LIN {X -0.008,Y -156.128,Z 1901.908,A 0.000,B 0.000,C 90.000,E1 343.378} C_DIS
LIN {X 0.025,Y -158.540,Z 1901.883,A 0.000,B 0.000,C 90.000,E1 338.901} C_DIS
LIN {X 0.039,Y -162.151,Z 1901.858,A 0.000,B 0.000,C 90.000,E1 334.460} C_DIS
LIN {X 0.090,Y -166.092,Z 1901.839,A 0.000,B 0.000,C 90.000,E1 330.923} C_DIS
LIN {X 0.023,Y -169.681,Z 1901.824,A 0.000,B 0.000,C 90.000,E1 328.329} C_DIS
LIN {X 0.058,Y -173.811,Z 1901.810,A 0.000,B 0.000,C 90.000,E1 325.722} C_DIS
LIN {X -0.019,Y -178.557,Z 1901.795,A 0.000,B 0.000,C 90.000,E1 323.176} C_DIS
LIN {X -0.047,Y -184.121,Z 1901.781,A 0.000,B 0.000,C 90.000,E1 320.642} C_DIS
LIN {X 0.007,Y -190.588,Z 1901.767,A 0.000,B 0.000,C 90.000,E1 318.119} C_DIS
LIN {X 0.021,Y -198.074,Z 1901.754,A 0.000,B 0.000,C 90.000,E1 315.648} C_DIS
LIN {X 0.040,Y -206.500,Z 1901.740,A 0.000,B 0.000,C 90.000,E1 313.218} C_DIS
LIN {X -0.005,Y -217.446,Z 1901.725,A 0.000,B 0.000,C 90.000,E1 310.458} C_DIS
LIN {X 0.024,Y -231.204,Z 1901.708,A 0.000,B 0.000,C 90.000,E1 307.363} C_DIS
LIN {X -0.156,Y -246.156,Z 1901.691,A 0.000,B 0.000,C 90.000,E1 304.405} C_DIS
LIN {X -0.150,Y -258.005,Z 1901.679,A 0.000,B 0.000,C 90.000,E1 302.212} C_DIS
LIN {X 0.093,Y -272.069,Z 1901.665,A 0.000,B 0.000,C 90.000,E1 299.667} C_DIS
LIN {X -0.131,Y -281.961,Z 1901.655,A 0.000,B 0.000,C 90.000,E1 297.975} C_DIS
LIN {X 0.044,Y -291.566,Z 1901.646,A 0.000,B 0.000,C 90.000,E1 296.232} C_DIS
LIN {X -0.014,Y -298.859,Z 1901.638,A 0.000,B 0.000,C 90.000,E1 294.899} C_DIS
LIN {X 0.154,Y -306.333,Z 1901.633,A 0.000,B 0.000,C 90.000,E1 293.823} C_DIS
LIN {X 0.160,Y -315.202,Z 1901.625,A 0.000,B 0.000,C 90.000,E1 292.514} C_DIS
LIN {X -0.072,Y -321.527,Z 1901.620,A 0.000,B 0.000,C 90.000,E1 291.589} C_DIS
LIN {X 0.003,Y -329.446,Z 1901.613,A 0.000,B 0.000,C 90.000,E1 290.301} C_DIS
LIN {X 0.047,Y -338.650,Z 1901.604,A 0.000,B 0.000,C 90.000,E1 288.725} C_DIS
LIN {X -0.090,Y -343.776,Z 1901.599,A 0.000,B 0.000,C 90.000,E1 287.819} C_DIS
LIN {X 0.146,Y -348.475,Z 1901.594,A 0.000,B 0.000,C 90.000,E1 286.858} C_DIS
LIN {X -0.001,Y -352.501,Z 1901.589,A 0.000,B 0.000,C 90.000,E1 285.969} C_DIS
LIN {X -0.022,Y -355.999,Z 1901.584,A 0.000,B 0.000,C 90.000,E1 285.064} C_DIS
LIN {X -0.140,Y -358.008,Z 1901.580,A 0.000,B 0.000,C 90.000,E1 284.481} C_DIS
LIN {X -0.161,Y -359.770,Z 1901.577,A 0.000,B 0.000,C 90.000,E1 283.883} C_DIS
LIN {X 0.094,Y -361.166,Z 1901.574,A 0.000,B 0.000,C 90.000,E1 283.244} C_DIS
LIN {X 0.093,Y -362.224,Z 1901.570,A 0.000,B 0.000,C 90.000,E1 282.647} C_DIS
LIN {X 0.017,Y -362.868,Z 1901.567,A 0.000,B 0.000,C 90.000,E1 282.063} C_DIS
LIN {X -0.050,Y -363.124,Z 1901.564,A 0.000,B 0.000,C 90.000,E1 281.478} C_DIS
LIN {X -0.113,Y -363.007,Z 1901.560,A 0.000,B 0.000,C 90.000,E1 280.894} C_DIS
LIN {X 0.182,Y -362.489,Z 1901.557,A 0.000,B 0.000,C 90.000,E1 280.254} C_DIS
LIN {X 0.117,Y -361.578,Z 1901.554,A 0.000,B 0.000,C 90.000,E1 279.670} C_DIS
LIN {X -0.008,Y -360.355,Z 1901.551,A 0.000,B 0.000,C 90.000,E1 279.095} C_DIS
LIN {X -0.081,Y -358.715,Z 1901.547,A 0.000,B 0.000,C 90.000,E1 278.511} C_DIS
LIN {X 0.093,Y -355.791,Z 1901.542,A 0.000,B 0.000,C 90.000,E1 277.587} C_DIS
LIN {X -0.112,Y -351.986,Z 1901.537,A 0.000,B 0.000,C 90.000,E1 276.720} C_DIS
LIN {X -0.007,Y -347.191,Z 1901.532,A 0.000,B 0.000,C 90.000,E1 275.796} C_DIS
LIN {X 0.141,Y -343.273,Z 1901.529,A 0.000,B 0.000,C 90.000,E1 275.163} C_DIS
LIN {X -0.075,Y -338.789,Z 1901.525,A 0.000,B 0.000,C 90.000,E1 274.588} C_DIS
LIN {X 0.022,Y -333.591,Z 1901.522,A 0.000,B 0.000,C 90.000,E1 273.955} C_DIS
LIN {X -0.141,Y -327.774,Z 1901.519,A 0.000,B 0.000,C 90.000,E1 273.383} C_DIS
LIN {X -0.062,Y -321.579,Z 1901.516,A 0.000,B 0.000,C 90.000,E1 272.808} C_DIS
LIN {X -0.009,Y -315.100,Z 1901.513,A 0.000,B 0.000,C 90.000,E1 272.293} C_DIS
LIN {X 0.118,Y -308.269,Z 1901.510,A 0.000,B 0.000,C 90.000,E1 271.835} C_DIS
LIN {X 0.007,Y -301.029,Z 1901.508,A 0.000,B 0.000,C 90.000,E1 271.489} C_DIS
LIN {X -0.028,Y -293.012,Z 1901.507,A 0.000,B 0.000,C 90.000,E1 271.203} C_DIS
LIN {X -0.091,Y -287.800,Z 1901.506,A 0.000,B 0.000,C 90.000,E1 271.088} C_DIS
LIN {X -0.114,Y -278.697,Z 1901.505,A 0.000,B 0.000,C 90.000,E1 270.974} C_DIS
LIN {X -0.029,Y -270.235,Z 1901.505,A 0.000,B 0.000,C 90.000,E1 270.917} C_DIS
LIN {X -0.041,Y -181.478,Z 1901.505,A 0.000,B 0.000,C 90.000,E1 270.917} C_DIS
LIN {X -0.028,Y -181.537,Z 1901.499,A 0.000,B 0.000,C 90.000,E1 269.885} C_DIS
LIN {X -0.085,Y -180.907,Z 1901.475,A 0.000,B 0.000,C 90.000,E1 265.527} C_DIS
LIN {X -0.027,Y -180.749,Z 1901.470,A 0.000,B 0.000,C 90.000,E1 264.666} C_DIS
LIN {X 0.041,Y -178.842,Z 1901.442,A 0.000,B 0.000,C 90.000,E1 259.577} C_DIS
LIN {X -0.063,Y -175.885,Z 1901.414,A 0.000,B 0.000,C 90.000,E1 254.519} C_DIS
LIN {X 0.044,Y -174.552,Z 1901.404,A 0.000,B 0.000,C 90.000,E1 252.779} C_DIS
LIN {X -0.025,Y -171.536,Z 1901.381,A 0.000,B 0.000,C 90.000,E1 248.518} C_DIS
LIN {X -0.031,Y -167.761,Z 1901.357,A 0.000,B 0.000,C 90.000,E1 244.204} C_DIS
LIN {X -0.088,Y -166.467,Z 1901.347,A 0.000,B 0.000,C 90.000,E1 242.487} C_DIS
LIN {X 0.048,Y -163.182,Z 1901.328,A 0.000,B 0.000,C 90.000,E1 238.948} C_DIS
LIN {X -0.037,Y -161.142,Z 1901.313,A 0.000,B 0.000,C 90.000,E1 236.342} C_DIS
LIN {X -0.001,Y -157.162,Z 1901.288,A 0.000,B 0.000,C 90.000,E1 231.904} C_DIS
LIN {X 0.022,Y -155.893,Z 1901.278,A 0.000,B 0.000,C 90.000,E1 230.114} C_DIS
LIN {X -0.020,Y -152.144,Z 1901.254,A 0.000,B 0.000,C 90.000,E1 225.648} C_DIS
LIN {X 0.000,Y -150.393,Z 1901.239,A 0.000,B 0.000,C 90.000,E1 222.933} C_DIS
LIN {X 0.024,Y -147.124,Z 1901.213,A 0.000,B 0.000,C 90.000,E1 218.382} C_DIS
LIN {X 0.015,Y -145.687,Z 1901.198,A 0.000,B 0.000,C 90.000,E1 215.644} C_DIS
LIN {X 0.013,Y -143.070,Z 1901.172,A 0.000,B 0.000,C 90.000,E1 211.052} C_DIS
LIN {X -0.056,Y -141.691,Z 1901.152,A 0.000,B 0.000,C 90.000,E1 207.385} C_DIS
LIN {X -0.002,Y -139.462,Z 1901.116,A 0.000,B 0.000,C 90.000,E1 200.865} C_DIS
LIN {X -0.033,Y -139.195,Z 1901.106,A 0.000,B 0.000,C 90.000,E1 199.014} C_DIS
LIN {X -0.015,Y -138.326,Z 1901.054,A 0.000,B 0.000,C 90.000,E1 189.670} C_DIS
LIN {X -0.010,Y -139.451,Z 1901.007,A 0.000,B 0.000,C 90.000,E1 181.260} C_DIS
LIN {X 0.070,Y -140.996,Z 1900.976,A 0.000,B 0.000,C 90.000,E1 175.641} C_DIS
LIN {X 0.020,Y -142.749,Z 1900.955,A 0.000,B 0.000,C 90.000,E1 171.951} C_DIS
LIN {X -0.024,Y -145.149,Z 1900.930,A 0.000,B 0.000,C 90.000,E1 167.353} C_DIS
LIN {X -0.031,Y -147.771,Z 1900.909,A 0.000,B 0.000,C 90.000,E1 163.685} C_DIS
LIN {X 0.049,Y -150.447,Z 1900.889,A 0.000,B 0.000,C 90.000,E1 160.007} C_DIS
LIN {X -0.017,Y -153.894,Z 1900.869,A 0.000,B 0.000,C 90.000,E1 156.410} C_DIS
LIN {X -0.023,Y -157.305,Z 1900.849,A 0.000,B 0.000,C 90.000,E1 152.820} C_DIS
LIN {X -0.004,Y -161.490,Z 1900.829,A 0.000,B 0.000,C 90.000,E1 149.253} C_DIS
LIN {X 0.011,Y -165.689,Z 1900.810,A 0.000,B 0.000,C 90.000,E1 145.722} C_DIS
LIN {X -0.102,Y -170.631,Z 1900.790,A 0.000,B 0.000,C 90.000,E1 142.271} C_DIS
LIN {X 0.052,Y -175.508,Z 1900.771,A 0.000,B 0.000,C 90.000,E1 138.771} C_DIS
LIN {X -0.082,Y -181.129,Z 1900.752,A 0.000,B 0.000,C 90.000,E1 135.405} C_DIS
LIN {X 0.045,Y -186.577,Z 1900.733,A 0.000,B 0.000,C 90.000,E1 132.000} C_DIS
LIN {X -0.006,Y -191.189,Z 1900.719,A 0.000,B 0.000,C 90.000,E1 129.519} C_DIS
LIN {X 0.040,Y -196.998,Z 1900.701,A 0.000,B 0.000,C 90.000,E1 126.217} C_DIS
LIN {X -0.042,Y -200.267,Z 1900.692,A 0.000,B 0.000,C 90.000,E1 124.612} C_DIS
LIN {X -0.049,Y -207.759,Z 1900.670,A 0.000,B 0.000,C 90.000,E1 120.590} C_DIS
LIN {X -0.046,Y -210.934,Z 1900.661,A 0.000,B 0.000,C 90.000,E1 118.999} C_DIS
LIN {X -0.040,Y -216.804,Z 1900.644,A 0.000,B 0.000,C 90.000,E1 115.848} C_DIS
LIN {X 0.108,Y -218.419,Z 1900.639,A 0.000,B 0.000,C 90.000,E1 115.027} C_DIS
LIN {X -0.053,Y -221.146,Z 1900.631,A 0.000,B 0.000,C 90.000,E1 113.515} C_DIS
LIN {X -0.062,Y -224.140,Z 1900.621,A 0.000,B 0.000,C 90.000,E1 111.844} C_DIS
LIN {X -0.111,Y -283.670,Z 1900.621,A 0.000,B 0.000,C 90.000,E1 111.844} C_DIS
LIN {X 0.092,Y -285.624,Z 1900.621,A 0.000,B 0.000,C 90.000,E1 111.770} C_DIS
LIN {X 0.027,Y -291.063,Z 1900.619,A 0.000,B 0.000,C 90.000,E1 111.482} C_DIS
LIN {X 0.066,Y -293.925,Z 1900.618,A 0.000,B 0.000,C 90.000,E1 111.173} C_DIS
LIN {X -0.146,Y -295.977,Z 1900.616,A 0.000,B 0.000,C 90.000,E1 110.918} C_DIS
LIN {X -0.054,Y -310.986,Z 1900.602,A 0.000,B 0.000,C 90.000,E1 108.290} C_DIS
LIN {X -0.018,Y -325.732,Z 1900.589,A 0.000,B 0.000,C 90.000,E1 106.024} C_DIS
LIN {X 0.068,Y -339.562,Z 1900.578,A 0.000,B 0.000,C 90.000,E1 104.120} C_DIS
LIN {X -0.082,Y -354.591,Z 1900.568,A 0.000,B 0.000,C 90.000,E1 102.299} C_DIS
LIN {X 0.090,Y -373.026,Z 1900.557,A 0.000,B 0.000,C 90.000,E1 100.254} C_DIS
LIN {X -0.167,Y -391.934,Z 1900.547,A 0.000,B 0.000,C 90.000,E1 98.454} C_DIS
LIN {X -0.127,Y -411.181,Z 1900.538,A 0.000,B 0.000,C 90.000,E1 96.777} C_DIS
LIN {X -0.181,Y -433.588,Z 1900.528,A 0.000,B 0.000,C 90.000,E1 95.049} C_DIS
LIN {X -0.202,Y -439.236,Z 1900.526,A 0.000,B 0.000,C 90.000,E1 94.645} C_DIS
LIN {X 0.011,Y -441.525,Z 1900.525,A 0.000,B 0.000,C 90.000,E1 94.416} C_DIS
LIN {X -0.022,Y -445.053,Z 1900.522,A 0.000,B 0.000,C 90.000,E1 93.955} C_DIS
LIN {X 0.151,Y -446.391,Z 1900.521,A 0.000,B 0.000,C 90.000,E1 93.669} C_DIS
LIN {X -0.120,Y -447.386,Z 1900.519,A 0.000,B 0.000,C 90.000,E1 93.440} C_DIS
LIN {X -0.163,Y -448.538,Z 1900.516,A 0.000,B 0.000,C 90.000,E1 92.922} C_DIS
LIN {X -0.223,Y -448.727,Z 1900.513,A 0.000,B 0.000,C 90.000,E1 92.407} C_DIS
LIN {X 0.176,Y -447.984,Z 1900.510,A 0.000,B 0.000,C 90.000,E1 91.835} C_DIS
LIN {X 0.140,Y -446.197,Z 1900.507,A 0.000,B 0.000,C 90.000,E1 91.318} C_DIS
LIN {X -0.109,Y -444.813,Z 1900.506,A 0.000,B 0.000,C 90.000,E1 91.088} C_DIS
LIN {X -0.021,Y -431.659,Z 1900.494,A 0.000,B 0.000,C 90.000,E1 88.969} C_DIS
LIN {X -0.041,Y -421.590,Z 1900.485,A 0.000,B 0.000,C 90.000,E1 87.364} C_DIS
LIN {X -0.125,Y -409.813,Z 1900.475,A 0.000,B 0.000,C 90.000,E1 85.469} C_DIS
LIN {X -0.057,Y -399.632,Z 1900.465,A 0.000,B 0.000,C 90.000,E1 83.799} C_DIS
LIN {X -0.119,Y -387.656,Z 1900.455,A 0.000,B 0.000,C 90.000,E1 81.837} C_DIS
LIN {X 0.076,Y -374.093,Z 1900.442,A 0.000,B 0.000,C 90.000,E1 79.511} C_DIS
LIN {X -0.009,Y -356.071,Z 1900.424,A 0.000,B 0.000,C 90.000,E1 76.284} C_DIS
LIN {X 0.010,Y -342.262,Z 1900.409,A 0.000,B 0.000,C 90.000,E1 73.559} C_DIS
LIN {X -0.031,Y -330.388,Z 1900.395,A 0.000,B 0.000,C 90.000,E1 71.094} C_DIS
LIN {X 0.098,Y -317.360,Z 1900.379,A 0.000,B 0.000,C 90.000,E1 68.230} C_DIS
LIN {X -0.076,Y -304.962,Z 1900.363,A 0.000,B 0.000,C 90.000,E1 65.357} C_DIS
LIN {X -0.057,Y -295.446,Z 1900.350,A 0.000,B 0.000,C 90.000,E1 63.050} C_DIS
LIN {X -0.111,Y -286.135,Z 1900.337,A 0.000,B 0.000,C 90.000,E1 60.717} C_DIS
LIN {X -0.085,Y -276.695,Z 1900.324,A 0.000,B 0.000,C 90.000,E1 58.329} C_DIS
LIN {X 0.012,Y -267.201,Z 1900.310,A 0.000,B 0.000,C 90.000,E1 55.881} C_DIS
LIN {X -0.020,Y -257.579,Z 1900.297,A 0.000,B 0.000,C 90.000,E1 53.417} C_DIS
LIN {X 0.042,Y -247.984,Z 1900.283,A 0.000,B 0.000,C 90.000,E1 50.884} C_DIS
LIN {X -0.005,Y -237.137,Z 1900.266,A 0.000,B 0.000,C 90.000,E1 47.957} C_DIS
LIN {X -0.021,Y -226.676,Z 1900.250,A 0.000,B 0.000,C 90.000,E1 44.960} C_DIS
LIN {X -0.056,Y -215.454,Z 1900.231,A 0.000,B 0.000,C 90.000,E1 41.515} C_DIS
LIN {X -0.080,Y -206.223,Z 1900.213,A 0.000,B 0.000,C 90.000,E1 38.382} C_DIS
LIN {X -0.068,Y -197.894,Z 1900.195,A 0.000,B 0.000,C 90.000,E1 35.185} C_DIS
LIN {X -0.046,Y -190.289,Z 1900.177,A 0.000,B 0.000,C 90.000,E1 31.926} C_DIS
LIN {X -0.030,Y -183.438,Z 1900.159,A 0.000,B 0.000,C 90.000,E1 28.615} C_DIS
LIN {X -0.113,Y -177.266,Z 1900.140,A 0.000,B 0.000,C 90.000,E1 25.283} C_DIS
LIN {X -0.007,Y -171.928,Z 1900.121,A 0.000,B 0.000,C 90.000,E1 21.844} C_DIS
LIN {X -0.067,Y -167.365,Z 1900.102,A 0.000,B 0.000,C 90.000,E1 18.417} C_DIS
LIN {X 0.033,Y -163.638,Z 1900.083,A 0.000,B 0.000,C 90.000,E1 14.898} C_DIS
LIN {X 0.064,Y -159.841,Z 1900.058,A 0.000,B 0.000,C 90.000,E1 10.489} C_DIS
LIN {X -0.028,Y -157.203,Z 1900.034,A 0.000,B 0.000,C 90.000,E1 6.087} C_DIS
LIN {X 0.000,Y -154.884,Z 1900.000,A 0.000,B 0.000,C 90.000,E1 360.000} C_DIS
LIN {X -0.012,Y -154.116,Z 1899.948,A 0.000,B 0.000,C 90.000,E1 350.557} C_DIS
LIN {X -0.008,Y -156.124,Z 1899.908,A 0.000,B 0.000,C 90.000,E1 343.378} C_DIS
LIN {X 0.025,Y -158.536,Z 1899.883,A 0.000,B 0.000,C 90.000,E1 338.901} C_DIS
LIN {X 0.038,Y -162.149,Z 1899.858,A 0.000,B 0.000,C 90.000,E1 334.460} C_DIS
LIN {X 0.089,Y -166.095,Z 1899.839,A 0.000,B 0.000,C 90.000,E1 330.923} C_DIS
LIN {X 0.023,Y -169.685,Z 1899.824,A 0.000,B 0.000,C 90.000,E1 328.329} C_DIS
LIN {X 0.056,Y -173.818,Z 1899.810,A 0.000,B 0.000,C 90.000,E1 325.722} C_DIS
LIN {X -0.019,Y -178.565,Z 1899.795,A 0.000,B 0.000,C 90.000,E1 323.176} C_DIS
LIN {X -0.047,Y -184.128,Z 1899.781,A 0.000,B 0.000,C 90.000,E1 320.642} C_DIS
LIN {X 0.007,Y -190.596,Z 1899.767,A 0.000,B 0.000,C 90.000,E1 318.119} C_DIS
LIN {X 0.020,Y -198.081,Z 1899.754,A 0.000,B 0.000,C 90.000,E1 315.648} C_DIS
LIN {X 0.040,Y -206.507,Z 1899.740,A 0.000,B 0.000,C 90.000,E1 313.218} C_DIS
LIN {X -0.005,Y -217.454,Z 1899.725,A 0.000,B 0.000,C 90.000,E1 310.458} C_DIS
LIN {X 0.024,Y -231.213,Z 1899.708,A 0.000,B 0.000,C 90.000,E1 307.363} C_DIS
LIN {X -0.155,Y -246.166,Z 1899.691,A 0.000,B 0.000,C 90.000,E1 304.405} C_DIS
LIN {X -0.150,Y -258.015,Z 1899.679,A 0.000,B 0.000,C 90.000,E1 302.212} C_DIS
LIN {X 0.093,Y -272.077,Z 1899.665,A 0.000,B 0.000,C 90.000,E1 299.667} C_DIS
LIN {X -0.130,Y -281.970,Z 1899.655,A 0.000,B 0.000,C 90.000,E1 297.975} C_DIS
LIN {X 0.045,Y -291.575,Z 1899.646,A 0.000,B 0.000,C 90.000,E1 296.232} C_DIS
LIN {X -0.129,Y -295.469,Z 1899.642,A 0.000,B 0.000,C 90.000,E1 295.591} C_DIS
LIN {X 0.060,Y -305.331,Z 1899.634,A 0.000,B 0.000,C 90.000,E1 294.131} C_DIS
LIN {X 0.048,Y -313.975,Z 1899.627,A 0.000,B 0.000,C 90.000,E1 292.823} C_DIS
LIN {X 0.029,Y -322.355,Z 1899.620,A 0.000,B 0.000,C 90.000,E1 291.535} C_DIS
LIN {X 0.119,Y -330.255,Z 1899.613,A 0.000,B 0.000,C 90.000,E1 290.248} C_DIS
LIN {X -0.139,Y -339.493,Z 1899.604,A 0.000,B 0.000,C 90.000,E1 288.725} C_DIS
LIN {X 0.057,Y -344.603,Z 1899.599,A 0.000,B 0.000,C 90.000,E1 287.764} C_DIS
LIN {X -0.037,Y -347.799,Z 1899.595,A 0.000,B 0.000,C 90.000,E1 287.166} C_DIS
LIN {X -0.097,Y -351.986,Z 1899.590,A 0.000,B 0.000,C 90.000,E1 286.260} C_DIS
LIN {X 0.129,Y -355.611,Z 1899.585,A 0.000,B 0.000,C 90.000,E1 285.315} C_DIS
LIN {X 0.047,Y -358.698,Z 1899.580,A 0.000,B 0.000,C 90.000,E1 284.426} C_DIS
LIN {X 0.031,Y -360.418,Z 1899.577,A 0.000,B 0.000,C 90.000,E1 283.828} C_DIS
LIN {X -0.059,Y -361.770,Z 1899.573,A 0.000,B 0.000,C 90.000,E1 283.244} C_DIS
LIN {X -0.057,Y -362.810,Z 1899.570,A 0.000,B 0.000,C 90.000,E1 282.647} C_DIS
LIN {X -0.129,Y -363.440,Z 1899.567,A 0.000,B 0.000,C 90.000,E1 282.063} C_DIS
LIN {X 0.164,Y -363.653,Z 1899.564,A 0.000,B 0.000,C 90.000,E1 281.422} C_DIS
LIN {X 0.104,Y -363.520,Z 1899.560,A 0.000,B 0.000,C 90.000,E1 280.838} C_DIS
LIN {X 0.045,Y -362.940,Z 1899.557,A 0.000,B 0.000,C 90.000,E1 280.254} C_DIS
LIN {X -0.015,Y -361.997,Z 1899.554,A 0.000,B 0.000,C 90.000,E1 279.670} C_DIS
LIN {X -0.138,Y -360.713,Z 1899.550,A 0.000,B 0.000,C 90.000,E1 279.095} C_DIS
LIN {X 0.147,Y -359.050,Z 1899.547,A 0.000,B 0.000,C 90.000,E1 278.454} C_DIS
LIN {X -0.029,Y -356.047,Z 1899.542,A 0.000,B 0.000,C 90.000,E1 277.587} C_DIS
LIN {X 0.120,Y -352.226,Z 1899.537,A 0.000,B 0.000,C 90.000,E1 276.663} C_DIS
LIN {X -0.122,Y -347.361,Z 1899.532,A 0.000,B 0.000,C 90.000,E1 275.796} C_DIS
LIN {X 0.029,Y -343.402,Z 1899.529,A 0.000,B 0.000,C 90.000,E1 275.163} C_DIS
LIN {X 0.153,Y -338.870,Z 1899.525,A 0.000,B 0.000,C 90.000,E1 274.531} C_DIS
LIN {X -0.084,Y -333.652,Z 1899.522,A 0.000,B 0.000,C 90.000,E1 273.955} C_DIS
LIN {X 0.106,Y -327.877,Z 1899.519,A 0.000,B 0.000,C 90.000,E1 273.326} C_DIS
LIN {X -0.085,Y -321.739,Z 1899.516,A 0.000,B 0.000,C 90.000,E1 272.808} C_DIS
LIN {X -0.012,Y -315.422,Z 1899.513,A 0.000,B 0.000,C 90.000,E1 272.293} C_DIS
LIN {X 0.059,Y -308.778,Z 1899.510,A 0.000,B 0.000,C 90.000,E1 271.835} C_DIS
LIN {X 0.150,Y -301.714,Z 1899.508,A 0.000,B 0.000,C 90.000,E1 271.432} C_DIS
LIN {X -0.007,Y -294.014,Z 1899.506,A 0.000,B 0.000,C 90.000,E1 271.146} C_DIS
LIN {X -0.027,Y -284.992,Z 1899.505,A 0.000,B 0.000,C 90.000,E1 270.917} C_DIS
LIN {X 0.132,Y -275.226,Z 1899.504,A 0.000,B 0.000,C 90.000,E1 270.745} C_DIS
LIN {X 0.093,Y -264.382,Z 1899.504,A 0.000,B 0.000,C 90.000,E1 270.688} C_DIS
LIN {X 0.034,Y -181.526,Z 1899.504,A 0.000,B 0.000,C 90.000,E1 270.688} C_DIS
LIN {X 0.084,Y -181.487,Z 1899.498,A 0.000,B 0.000,C 90.000,E1 269.656} C_DIS
LIN {X 0.026,Y -180.904,Z 1899.474,A 0.000,B 0.000,C 90.000,E1 265.298} C_DIS
LIN {X -0.024,Y -180.247,Z 1899.465,A 0.000,B 0.000,C 90.000,E1 263.628} C_DIS
LIN {X -0.005,Y -178.736,Z 1899.441,A 0.000,B 0.000,C 90.000,E1 259.398} C_DIS
LIN {X 0.061,Y -175.784,Z 1899.413,A 0.000,B 0.000,C 90.000,E1 254.283} C_DIS
LIN {X 0.049,Y -171.968,Z 1899.384,A 0.000,B 0.000,C 90.000,E1 249.156} C_DIS
LIN {X 0.087,Y -171.366,Z 1899.380,A 0.000,B 0.000,C 90.000,E1 248.284} C_DIS
LIN {X -0.088,Y -167.614,Z 1899.355,A 0.000,B 0.000,C 90.000,E1 244.024} C_DIS
LIN {X 0.076,Y -166.263,Z 1899.346,A 0.000,B 0.000,C 90.000,E1 242.231} C_DIS
LIN {X 0.063,Y -163.016,Z 1899.326,A 0.000,B 0.000,C 90.000,E1 238.742} C_DIS
LIN {X -0.024,Y -160.940,Z 1899.312,A 0.000,B 0.000,C 90.000,E1 236.135} C_DIS
LIN {X 0.085,Y -157.698,Z 1899.292,A 0.000,B 0.000,C 90.000,E1 232.557} C_DIS
LIN {X 0.024,Y -155.738,Z 1899.277,A 0.000,B 0.000,C 90.000,E1 229.908} C_DIS
LIN {X 0.077,Y -151.996,Z 1899.252,A 0.000,B 0.000,C 90.000,E1 225.405} C_DIS
LIN {X 0.092,Y -150.241,Z 1899.237,A 0.000,B 0.000,C 90.000,E1 222.690} C_DIS
LIN {X 0.015,Y -147.000,Z 1899.212,A 0.000,B 0.000,C 90.000,E1 218.177} C_DIS
LIN {X 0.005,Y -145.584,Z 1899.197,A 0.000,B 0.000,C 90.000,E1 215.438} C_DIS
LIN {X -0.001,Y -142.973,Z 1899.171,A 0.000,B 0.000,C 90.000,E1 210.846} C_DIS
LIN {X 0.052,Y -141.600,Z 1899.151,A 0.000,B 0.000,C 90.000,E1 207.129} C_DIS
LIN {X -0.032,Y -139.423,Z 1899.115,A 0.000,B 0.000,C 90.000,E1 200.663} C_DIS
LIN {X 0.019,Y -139.150,Z 1899.104,A 0.000,B 0.000,C 90.000,E1 198.779} C_DIS
LIN {X 0.041,Y -138.344,Z 1899.058,A 0.000,B 0.000,C 90.000,E1 190.366} C_DIS
LIN {X 0.027,Y -139.486,Z 1899.006,A 0.000,B 0.000,C 90.000,E1 181.031} C_DIS
LIN {X -0.033,Y -141.084,Z 1898.975,A 0.000,B 0.000,C 90.000,E1 175.469} C_DIS
LIN {X 0.061,Y -142.461,Z 1898.959,A 0.000,B 0.000,C 90.000,E1 172.648} C_DIS
LIN {X 0.010,Y -144.706,Z 1898.934,A 0.000,B 0.000,C 90.000,E1 168.049} C_DIS
LIN {X -0.038,Y -147.303,Z 1898.913,A 0.000,B 0.000,C 90.000,E1 164.393} C_DIS
LIN {X -0.024,Y -150.624,Z 1898.888,A 0.000,B 0.000,C 90.000,E1 159.826} C_DIS
LIN {X 0.053,Y -154.099,Z 1898.868,A 0.000,B 0.000,C 90.000,E1 156.177} C_DIS
LIN {X -0.023,Y -157.522,Z 1898.848,A 0.000,B 0.000,C 90.000,E1 152.615} C_DIS
LIN {X -0.079,Y -161.756,Z 1898.828,A 0.000,B 0.000,C 90.000,E1 149.076} C_DIS
LIN {X 0.027,Y -165.949,Z 1898.808,A 0.000,B 0.000,C 90.000,E1 145.515} C_DIS
LIN {X 0.024,Y -170.940,Z 1898.789,A 0.000,B 0.000,C 90.000,E1 142.029} C_DIS
LIN {X -0.056,Y -175.809,Z 1898.770,A 0.000,B 0.000,C 90.000,E1 138.609} C_DIS
LIN {X 0.072,Y -181.416,Z 1898.751,A 0.000,B 0.000,C 90.000,E1 135.162} C_DIS
LIN {X -0.053,Y -186.918,Z 1898.732,A 0.000,B 0.000,C 90.000,E1 131.838} C_DIS
LIN {X 0.020,Y -191.497,Z 1898.719,A 0.000,B 0.000,C 90.000,E1 129.322} C_DIS
LIN {X 0.105,Y -197.361,Z 1898.700,A 0.000,B 0.000,C 90.000,E1 126.011} C_DIS
LIN {X 0.030,Y -200.637,Z 1898.691,A 0.000,B 0.000,C 90.000,E1 124.405} C_DIS
LIN {X -0.060,Y -206.521,Z 1898.673,A 0.000,B 0.000,C 90.000,E1 121.209} C_DIS
LIN {X 0.034,Y -209.811,Z 1898.664,A 0.000,B 0.000,C 90.000,E1 119.589} C_DIS
LIN {X -0.040,Y -217.169,Z 1898.643,A 0.000,B 0.000,C 90.000,E1 115.668} C_DIS
LIN {X -0.085,Y -218.796,Z 1898.638,A 0.000,B 0.000,C 90.000,E1 114.899} C_DIS
LIN {X -0.069,Y -224.144,Z 1898.621,A 0.000,B 0.000,C 90.000,E1 111.844} C_DIS
LIN {X -0.121,Y -284.036,Z 1898.621,A 0.000,B 0.000,C 90.000,E1 111.844} C_DIS
LIN {X 0.048,Y -285.983,Z 1898.621,A 0.000,B 0.000,C 90.000,E1 111.770} C_DIS
LIN {X 0.130,Y -289.404,Z 1898.620,A 0.000,B 0.000,C 90.000,E1 111.589} C_DIS
LIN {X 0.176,Y -292.839,Z 1898.618,A 0.000,B 0.000,C 90.000,E1 111.280} C_DIS
LIN {X 0.071,Y -296.478,Z 1898.616,A 0.000,B 0.000,C 90.000,E1 110.791} C_DIS
LIN {X -0.031,Y -309.743,Z 1898.603,A 0.000,B 0.000,C 90.000,E1 108.489} C_DIS
LIN {X 0.080,Y -324.361,Z 1898.590,A 0.000,B 0.000,C 90.000,E1 106.205} C_DIS
LIN {X 0.146,Y -338.072,Z 1898.580,A 0.000,B 0.000,C 90.000,E1 104.300} C_DIS
LIN {X -0.025,Y -352.972,Z 1898.569,A 0.000,B 0.000,C 90.000,E1 102.479} C_DIS
LIN {X 0.041,Y -371.365,Z 1898.558,A 0.000,B 0.000,C 90.000,E1 100.433} C_DIS
LIN {X 0.127,Y -390.236,Z 1898.548,A 0.000,B 0.000,C 90.000,E1 98.568} C_DIS
LIN {X 0.082,Y -409.450,Z 1898.538,A 0.000,B 0.000,C 90.000,E1 96.891} C_DIS
LIN {X -0.071,Y -431.829,Z 1898.529,A 0.000,B 0.000,C 90.000,E1 95.163} C_DIS
LIN {X 0.085,Y -440.191,Z 1898.525,A 0.000,B 0.000,C 90.000,E1 94.531} C_DIS
LIN {X -0.031,Y -443.932,Z 1898.523,A 0.000,B 0.000,C 90.000,E1 94.131} C_DIS
LIN {X 0.169,Y -445.542,Z 1898.521,A 0.000,B 0.000,C 90.000,E1 93.841} C_DIS
LIN {X -0.106,Y -446.756,Z 1898.520,A 0.000,B 0.000,C 90.000,E1 93.612} C_DIS
LIN {X -0.154,Y -448.257,Z 1898.517,A 0.000,B 0.000,C 90.000,E1 93.094} C_DIS
LIN {X -0.218,Y -448.753,Z 1898.514,A 0.000,B 0.000,C 90.000,E1 92.579} C_DIS
LIN {X 0.178,Y -448.320,Z 1898.511,A 0.000,B 0.000,C 90.000,E1 92.007} C_DIS
LIN {X 0.143,Y -446.901,Z 1898.508,A 0.000,B 0.000,C 90.000,E1 91.489} C_DIS
LIN {X -0.106,Y -445.751,Z 1898.507,A 0.000,B 0.000,C 90.000,E1 91.260} C_DIS
LIN {X 0.205,Y -439.284,Z 1898.501,A 0.000,B 0.000,C 90.000,E1 90.172} C_DIS
LIN {X -0.125,Y -429.425,Z 1898.492,A 0.000,B 0.000,C 90.000,E1 88.625} C_DIS
LIN {X -0.050,Y -417.625,Z 1898.482,A 0.000,B 0.000,C 90.000,E1 86.731} C_DIS
LIN {X 0.189,Y -405.837,Z 1898.471,A 0.000,B 0.000,C 90.000,E1 84.780} C_DIS
LIN {X -0.140,Y -393.895,Z 1898.460,A 0.000,B 0.000,C 90.000,E1 82.875} C_DIS
LIN {X 0.115,Y -381.954,Z 1898.449,A 0.000,B 0.000,C 90.000,E1 80.849} C_DIS
LIN {X 0.168,Y -368.450,Z 1898.436,A 0.000,B 0.000,C 90.000,E1 78.522} C_DIS
LIN {X 0.030,Y -352.386,Z 1898.420,A 0.000,B 0.000,C 90.000,E1 75.574} C_DIS
LIN {X 0.047,Y -338.733,Z 1898.405,A 0.000,B 0.000,C 90.000,E1 72.834} C_DIS
LIN {X -0.078,Y -326.939,Z 1898.391,A 0.000,B 0.000,C 90.000,E1 70.369} C_DIS
LIN {X -0.006,Y -312.664,Z 1898.373,A 0.000,B 0.000,C 90.000,E1 67.177} C_DIS
LIN {X -0.065,Y -301.772,Z 1898.359,A 0.000,B 0.000,C 90.000,E1 64.588} C_DIS
LIN {X -0.009,Y -289.633,Z 1898.342,A 0.000,B 0.000,C 90.000,E1 61.591} C_DIS
LIN {X 0.116,Y -281.614,Z 1898.331,A 0.000,B 0.000,C 90.000,E1 59.537} C_DIS
LIN {X -0.055,Y -272.131,Z 1898.318,A 0.000,B 0.000,C 90.000,E1 57.168} C_DIS
LIN {X 0.027,Y -263.959,Z 1898.306,A 0.000,B 0.000,C 90.000,E1 55.055} C_DIS
LIN {X 0.071,Y -254.351,Z 1898.292,A 0.000,B 0.000,C 90.000,E1 52.557} C_DIS
LIN {X 0.027,Y -244.761,Z 1898.278,A 0.000,B 0.000,C 90.000,E1 50.033} C_DIS
LIN {X 0.066,Y -233.998,Z 1898.262,A 0.000,B 0.000,C 90.000,E1 47.067} C_DIS
LIN {X 0.134,Y -223.664,Z 1898.245,A 0.000,B 0.000,C 90.000,E1 44.028} C_DIS
LIN {X -0.129,Y -212.650,Z 1898.225,A 0.000,B 0.000,C 90.000,E1 40.620} C_DIS
LIN {X 0.057,Y -204.730,Z 1898.210,A 0.000,B 0.000,C 90.000,E1 37.810} C_DIS
LIN {X 0.028,Y -196.532,Z 1898.192,A 0.000,B 0.000,C 90.000,E1 34.612} C_DIS
LIN {X 0.070,Y -189.066,Z 1898.174,A 0.000,B 0.000,C 90.000,E1 31.337} C_DIS
LIN {X 0.053,Y -182.332,Z 1898.156,A 0.000,B 0.000,C 90.000,E1 28.025} C_DIS
LIN {X 0.099,Y -176.297,Z 1898.137,A 0.000,B 0.000,C 90.000,E1 24.643} C_DIS
LIN {X -0.053,Y -171.096,Z 1898.118,A 0.000,B 0.000,C 90.000,E1 21.280} C_DIS
LIN {X -0.032,Y -166.675,Z 1898.099,A 0.000,B 0.000,C 90.000,E1 17.819} C_DIS
LIN {X 0.052,Y -163.066,Z 1898.080,A 0.000,B 0.000,C 90.000,E1 14.300} C_DIS
LIN {X 0.028,Y -159.406,Z 1898.055,A 0.000,B 0.000,C 90.000,E1 9.905} C_DIS
LIN {X 0.058,Y -156.925,Z 1898.030,A 0.000,B 0.000,C 90.000,E1 5.454} C_DIS
LIN {X 0.026,Y -154.529,Z 1897.992,A 0.000,B 0.000,C 90.000,E1 358.625} C_DIS
LIN {X 0.004,Y -155.157,Z 1897.923,A 0.000,B 0.000,C 90.000,E1 346.061} C_DIS
LIN {X 0.042,Y -157.434,Z 1897.893,A 0.000,B 0.000,C 90.000,E1 340.678} C_DIS
LIN {X 0.039,Y -160.568,Z 1897.868,A 0.000,B 0.000,C 90.000,E1 336.230} C_DIS
LIN {X -0.095,Y -163.996,Z 1897.848,A 0.000,B 0.000,C 90.000,E1 332.743} C_DIS
LIN {X 0.008,Y -168.423,Z 1897.829,A 0.000,B 0.000,C 90.000,E1 329.203} C_DIS
LIN {X 0.055,Y -173.824,Z 1897.810,A 0.000,B 0.000,C 90.000,E1 325.722} C_DIS
LIN {X -0.021,Y -178.573,Z 1897.795,A 0.000,B 0.000,C 90.000,E1 323.176} C_DIS
LIN {X -0.048,Y -184.137,Z 1897.781,A 0.000,B 0.000,C 90.000,E1 320.642} C_DIS
LIN {X 0.006,Y -190.605,Z 1897.767,A 0.000,B 0.000,C 90.000,E1 318.119} C_DIS
LIN {X 0.020,Y -198.086,Z 1897.754,A 0.000,B 0.000,C 90.000,E1 315.648} C_DIS
LIN {X 0.040,Y -206.512,Z 1897.740,A 0.000,B 0.000,C 90.000,E1 313.218} C_DIS
LIN {X -0.006,Y -217.461,Z 1897.725,A 0.000,B 0.000,C 90.000,E1 310.458} C_DIS
LIN {X 0.024,Y -231.221,Z 1897.708,A 0.000,B 0.000,C 90.000,E1 307.363} C_DIS
LIN {X -0.155,Y -246.176,Z 1897.691,A 0.000,B 0.000,C 90.000,E1 304.405} C_DIS
LIN {X -0.150,Y -258.025,Z 1897.679,A 0.000,B 0.000,C 90.000,E1 302.212} C_DIS
LIN {X 0.094,Y -272.086,Z 1897.665,A 0.000,B 0.000,C 90.000,E1 299.667} C_DIS
LIN {X -0.130,Y -281.978,Z 1897.655,A 0.000,B 0.000,C 90.000,E1 297.975} C_DIS
LIN {X 0.077,Y -289.696,Z 1897.648,A 0.000,B 0.000,C 90.000,E1 296.565} C_DIS
LIN {X 0.043,Y -301.749,Z 1897.638,A 0.000,B 0.000,C 90.000,E1 294.771} C_DIS
LIN {X -0.011,Y -310.447,Z 1897.630,A 0.000,B 0.000,C 90.000,E1 293.462} C_DIS
LIN {X -0.031,Y -320.992,Z 1897.621,A 0.000,B 0.000,C 90.000,E1 291.844} C_DIS
LIN {X 0.042,Y -329.046,Z 1897.614,A 0.000,B 0.000,C 90.000,E1 290.556} C_DIS
LIN {X 0.202,Y -338.470,Z 1897.605,A 0.000,B 0.000,C 90.000,E1 288.960} C_DIS
LIN {X -0.045,Y -345.380,Z 1897.599,A 0.000,B 0.000,C 90.000,E1 287.764} C_DIS
LIN {X -0.034,Y -348.552,Z 1897.595,A 0.000,B 0.000,C 90.000,E1 287.149} C_DIS
LIN {X 0.148,Y -352.681,Z 1897.590,A 0.000,B 0.000,C 90.000,E1 286.205} C_DIS
LIN {X 0.042,Y -356.299,Z 1897.585,A 0.000,B 0.000,C 90.000,E1 285.315} C_DIS
LIN {X -0.035,Y -359.350,Z 1897.580,A 0.000,B 0.000,C 90.000,E1 284.426} C_DIS
LIN {X -0.047,Y -361.034,Z 1897.577,A 0.000,B 0.000,C 90.000,E1 283.828} C_DIS
LIN {X -0.133,Y -362.395,Z 1897.573,A 0.000,B 0.000,C 90.000,E1 283.244} C_DIS
LIN {X -0.128,Y -363.399,Z 1897.570,A 0.000,B 0.000,C 90.000,E1 282.647} C_DIS
LIN {X 0.160,Y -363.978,Z 1897.567,A 0.000,B 0.000,C 90.000,E1 282.007} C_DIS
LIN {X 0.101,Y -364.167,Z 1897.564,A 0.000,B 0.000,C 90.000,E1 281.422} C_DIS
LIN {X 0.044,Y -364.016,Z 1897.560,A 0.000,B 0.000,C 90.000,E1 280.838} C_DIS
LIN {X -0.011,Y -363.403,Z 1897.557,A 0.000,B 0.000,C 90.000,E1 280.254} C_DIS
LIN {X -0.069,Y -362.427,Z 1897.554,A 0.000,B 0.000,C 90.000,E1 279.670} C_DIS
LIN {X -0.132,Y -361.100,Z 1897.550,A 0.000,B 0.000,C 90.000,E1 279.086} C_DIS
LIN {X 0.099,Y -359.425,Z 1897.547,A 0.000,B 0.000,C 90.000,E1 278.454} C_DIS
LIN {X -0.073,Y -356.359,Z 1897.542,A 0.000,B 0.000,C 90.000,E1 277.587} C_DIS
LIN {X 0.080,Y -352.506,Z 1897.537,A 0.000,B 0.000,C 90.000,E1 276.663} C_DIS
LIN {X -0.086,Y -349.311,Z 1897.534,A 0.000,B 0.000,C 90.000,E1 276.087} C_DIS
LIN {X 0.079,Y -345.674,Z 1897.530,A 0.000,B 0.000,C 90.000,E1 275.454} C_DIS
LIN {X -0.122,Y -341.402,Z 1897.527,A 0.000,B 0.000,C 90.000,E1 274.878} C_DIS
LIN {X -0.005,Y -336.507,Z 1897.524,A 0.000,B 0.000,C 90.000,E1 274.245} C_DIS
LIN {X 0.080,Y -330.889,Z 1897.520,A 0.000,B 0.000,C 90.000,E1 273.612} C_DIS
LIN {X 0.057,Y -324.870,Z 1897.517,A 0.000,B 0.000,C 90.000,E1 273.037} C_DIS
LIN {X -0.009,Y -318.556,Z 1897.514,A 0.000,B 0.000,C 90.000,E1 272.522} C_DIS
LIN {X -0.072,Y -312.163,Z 1897.511,A 0.000,B 0.000,C 90.000,E1 272.064} C_DIS
LIN {X 0.149,Y -305.349,Z 1897.509,A 0.000,B 0.000,C 90.000,E1 271.604} C_DIS
LIN {X 0.048,Y -298.180,Z 1897.507,A 0.000,B 0.000,C 90.000,E1 271.260} C_DIS
LIN {X -0.015,Y -290.063,Z 1897.505,A 0.000,B 0.000,C 90.000,E1 270.974} C_DIS
LIN {X 0.073,Y -281.028,Z 1897.504,A 0.000,B 0.000,C 90.000,E1 270.745} C_DIS
LIN {X -0.067,Y -271.247,Z 1897.503,A 0.000,B 0.000,C 90.000,E1 270.630} C_DIS
LIN {X 0.013,Y -258.848,Z 1897.503,A 0.000,B 0.000,C 90.000,E1 270.516} C_DIS
LIN {X -0.036,Y -255.801,Z 1897.503,A 0.000,B 0.000,C 90.000,E1 270.516} C_DIS
LIN {X -0.061,Y -181.566,Z 1897.503,A 0.000,B 0.000,C 90.000,E1 270.516} C_DIS
LIN {X 0.041,Y -181.116,Z 1897.489,A 0.000,B 0.000,C 90.000,E1 267.936} C_DIS
LIN {X 0.030,Y -180.906,Z 1897.475,A 0.000,B 0.000,C 90.000,E1 265.412} C_DIS
LIN {X -0.094,Y -180.714,Z 1897.470,A 0.000,B 0.000,C 90.000,E1 264.609} C_DIS
LIN {X 0.004,Y -178.801,Z 1897.442,A 0.000,B 0.000,C 90.000,E1 259.511} C_DIS
LIN {X 0.081,Y -175.847,Z 1897.413,A 0.000,B 0.000,C 90.000,E1 254.393} C_DIS
LIN {X 0.041,Y -172.582,Z 1897.390,A 0.000,B 0.000,C 90.000,E1 250.134} C_DIS
LIN {X 0.056,Y -171.470,Z 1897.380,A 0.000,B 0.000,C 90.000,E1 248.411} C_DIS
LIN {X 0.036,Y -167.702,Z 1897.356,A 0.000,B 0.000,C 90.000,E1 244.101} C_DIS
LIN {X 0.049,Y -166.387,Z 1897.347,A 0.000,B 0.000,C 90.000,E1 242.359} C_DIS
LIN {X 0.041,Y -163.114,Z 1897.327,A 0.000,B 0.000,C 90.000,E1 238.869} C_DIS
LIN {X 0.091,Y -161.063,Z 1897.313,A 0.000,B 0.000,C 90.000,E1 236.215} C_DIS
LIN {X -0.023,Y -157.797,Z 1897.293,A 0.000,B 0.000,C 90.000,E1 232.718} C_DIS
LIN {X 0.017,Y -155.833,Z 1897.278,A 0.000,B 0.000,C 90.000,E1 230.033} C_DIS
LIN {X -0.026,Y -152.083,Z 1897.253,A 0.000,B 0.000,C 90.000,E1 225.567} C_DIS
LIN {X -0.008,Y -150.334,Z 1897.238,A 0.000,B 0.000,C 90.000,E1 222.852} C_DIS
LIN {X 0.014,Y -147.073,Z 1897.213,A 0.000,B 0.000,C 90.000,E1 218.302} C_DIS
LIN {X -0.083,Y -145.648,Z 1897.198,A 0.000,B 0.000,C 90.000,E1 215.598} C_DIS
LIN {X -0.079,Y -143.030,Z 1897.172,A 0.000,B 0.000,C 90.000,E1 211.003} C_DIS
LIN {X 0.049,Y -141.656,Z 1897.151,A 0.000,B 0.000,C 90.000,E1 207.257} C_DIS
LIN {X -0.032,Y -139.446,Z 1897.115,A 0.000,B 0.000,C 90.000,E1 200.791} C_DIS
LIN {X 0.021,Y -139.179,Z 1897.105,A 0.000,B 0.000,C 90.000,E1 198.906} C_DIS
LIN {X 0.049,Y -138.320,Z 1897.053,A 0.000,B 0.000,C 90.000,E1 189.557} C_DIS
LIN {X 0.058,Y -139.466,Z 1897.006,A 0.000,B 0.000,C 90.000,E1 181.146} C_DIS
LIN {X -0.001,Y -141.031,Z 1896.975,A 0.000,B 0.000,C 90.000,E1 175.584} C_DIS
LIN {X -0.047,Y -142.398,Z 1896.960,A 0.000,B 0.000,C 90.000,E1 172.818} C_DIS
LIN {X 0.016,Y -144.630,Z 1896.934,A 0.000,B 0.000,C 90.000,E1 168.173} C_DIS
LIN {X 0.075,Y -147.825,Z 1896.909,A 0.000,B 0.000,C 90.000,E1 163.559} C_DIS
LIN {X 0.020,Y -150.518,Z 1896.889,A 0.000,B 0.000,C 90.000,E1 159.934} C_DIS
LIN {X 0.041,Y -153.979,Z 1896.868,A 0.000,B 0.000,C 90.000,E1 156.305} C_DIS
LIN {X -0.039,Y -157.392,Z 1896.849,A 0.000,B 0.000,C 90.000,E1 152.743} C_DIS
LIN {X 0.041,Y -161.597,Z 1896.829,A 0.000,B 0.000,C 90.000,E1 149.154} C_DIS
LIN {X -0.087,Y -165.794,Z 1896.809,A 0.000,B 0.000,C 90.000,E1 145.674} C_DIS
LIN {X 0.033,Y -170.756,Z 1896.790,A 0.000,B 0.000,C 90.000,E1 142.145} C_DIS
LIN {X 0.056,Y -175.628,Z 1896.771,A 0.000,B 0.000,C 90.000,E1 138.690} C_DIS
LIN {X -0.074,Y -181.245,Z 1896.752,A 0.000,B 0.000,C 90.000,E1 135.324} C_DIS
LIN {X 0.056,Y -186.715,Z 1896.733,A 0.000,B 0.000,C 90.000,E1 131.919} C_DIS
LIN {X 0.007,Y -191.314,Z 1896.719,A 0.000,B 0.000,C 90.000,E1 129.439} C_DIS
LIN {X -0.062,Y -197.144,Z 1896.701,A 0.000,B 0.000,C 90.000,E1 126.171} C_DIS
LIN {X -0.027,Y -200.420,Z 1896.692,A 0.000,B 0.000,C 90.000,E1 124.532} C_DIS
LIN {X -0.126,Y -206.304,Z 1896.674,A 0.000,B 0.000,C 90.000,E1 121.337} C_DIS
LIN {X -0.036,Y -209.578,Z 1896.665,A 0.000,B 0.000,C 90.000,E1 119.716} C_DIS
LIN {X 0.032,Y -215.391,Z 1896.647,A 0.000,B 0.000,C 90.000,E1 116.539} C_DIS
LIN {X 0.031,Y -218.572,Z 1896.639,A 0.000,B 0.000,C 90.000,E1 114.975} C_DIS
LIN {X -0.065,Y -224.142,Z 1896.621,A 0.000,B 0.000,C 90.000,E1 111.844} C_DIS
LIN {X -0.117,Y -284.090,Z 1896.621,A 0.000,B 0.000,C 90.000,E1 111.844} C_DIS
LIN {X 0.042,Y -285.289,Z 1896.621,A 0.000,B 0.000,C 90.000,E1 111.791} C_DIS
LIN {X -0.069,Y -289.205,Z 1896.620,A 0.000,B 0.000,C 90.000,E1 111.642} C_DIS
LIN {X -0.019,Y -291.419,Z 1896.619,A 0.000,B 0.000,C 90.000,E1 111.461} C_DIS
LIN {X 0.082,Y -294.473,Z 1896.617,A 0.000,B 0.000,C 90.000,E1 111.099} C_DIS
LIN {X 0.070,Y -296.479,Z 1896.616,A 0.000,B 0.000,C 90.000,E1 110.791} C_DIS
LIN {X 0.103,Y -309.591,Z 1896.603,A 0.000,B 0.000,C 90.000,E1 108.489} C_DIS
LIN {X -0.089,Y -324.186,Z 1896.590,A 0.000,B 0.000,C 90.000,E1 106.260} C_DIS
LIN {X -0.035,Y -337.882,Z 1896.580,A 0.000,B 0.000,C 90.000,E1 104.356} C_DIS
LIN {X 0.125,Y -352.764,Z 1896.569,A 0.000,B 0.000,C 90.000,E1 102.479} C_DIS
LIN {X -0.201,Y -371.180,Z 1896.558,A 0.000,B 0.000,C 90.000,E1 100.489} C_DIS
LIN {X -0.118,Y -390.010,Z 1896.548,A 0.000,B 0.000,C 90.000,E1 98.624} C_DIS
LIN {X 0.195,Y -409.257,Z 1896.538,A 0.000,B 0.000,C 90.000,E1 96.891} C_DIS
LIN {X 0.038,Y -431.630,Z 1896.529,A 0.000,B 0.000,C 90.000,E1 95.163} C_DIS
LIN {X 0.212,Y -439.992,Z 1896.525,A 0.000,B 0.000,C 90.000,E1 94.531} C_DIS
LIN {X -0.010,Y -442.078,Z 1896.524,A 0.000,B 0.000,C 90.000,E1 94.359} C_DIS
LIN {X -0.151,Y -444.032,Z 1896.523,A 0.000,B 0.000,C 90.000,E1 94.131} C_DIS
LIN {X 0.182,Y -445.524,Z 1896.521,A 0.000,B 0.000,C 90.000,E1 93.841} C_DIS
LIN {X -0.082,Y -446.732,Z 1896.520,A 0.000,B 0.000,C 90.000,E1 93.612} C_DIS
LIN {X 0.101,Y -447.625,Z 1896.519,A 0.000,B 0.000,C 90.000,E1 93.326} C_DIS
LIN {X 0.061,Y -448.607,Z 1896.516,A 0.000,B 0.000,C 90.000,E1 92.808} C_DIS
LIN {X 0.004,Y -448.640,Z 1896.513,A 0.000,B 0.000,C 90.000,E1 92.293} C_DIS
LIN {X -0.031,Y -447.736,Z 1896.510,A 0.000,B 0.000,C 90.000,E1 91.776} C_DIS
LIN {X -0.081,Y -445.750,Z 1896.507,A 0.000,B 0.000,C 90.000,E1 91.260} C_DIS
LIN {X -0.205,Y -439.289,Z 1896.501,A 0.000,B 0.000,C 90.000,E1 90.229} C_DIS
LIN {X -0.097,Y -429.429,Z 1896.492,A 0.000,B 0.000,C 90.000,E1 88.625} C_DIS
LIN {X -0.026,Y -417.627,Z 1896.482,A 0.000,B 0.000,C 90.000,E1 86.731} C_DIS
LIN {X -0.188,Y -405.843,Z 1896.471,A 0.000,B 0.000,C 90.000,E1 84.837} C_DIS
LIN {X -0.119,Y -393.896,Z 1896.460,A 0.000,B 0.000,C 90.000,E1 82.875} C_DIS
LIN {X 0.141,Y -381.959,Z 1896.449,A 0.000,B 0.000,C 90.000,E1 80.849} C_DIS
LIN {X -0.168,Y -368.454,Z 1896.436,A 0.000,B 0.000,C 90.000,E1 78.578} C_DIS
LIN {X -0.034,Y -352.388,Z 1896.420,A 0.000,B 0.000,C 90.000,E1 75.589} C_DIS
LIN {X -0.035,Y -338.730,Z 1896.405,A 0.000,B 0.000,C 90.000,E1 72.851} C_DIS
LIN {X -0.060,Y -326.932,Z 1896.391,A 0.000,B 0.000,C 90.000,E1 70.369} C_DIS
LIN {X 0.011,Y -312.658,Z 1896.373,A 0.000,B 0.000,C 90.000,E1 67.177} C_DIS
LIN {X -0.049,Y -301.763,Z 1896.359,A 0.000,B 0.000,C 90.000,E1 64.588} C_DIS
LIN {X 0.011,Y -289.625,Z 1896.342,A 0.000,B 0.000,C 90.000,E1 61.591} C_DIS
LIN {X 0.135,Y -281.607,Z 1896.331,A 0.000,B 0.000,C 90.000,E1 59.537} C_DIS
LIN {X -0.042,Y -272.121,Z 1896.318,A 0.000,B 0.000,C 90.000,E1 57.168} C_DIS
LIN {X 0.041,Y -263.952,Z 1896.306,A 0.000,B 0.000,C 90.000,E1 55.055} C_DIS
LIN {X 0.088,Y -254.347,Z 1896.292,A 0.000,B 0.000,C 90.000,E1 52.557} C_DIS
LIN {X -0.117,Y -244.755,Z 1896.278,A 0.000,B 0.000,C 90.000,E1 50.070} C_DIS
LIN {X 0.076,Y -233.990,Z 1896.262,A 0.000,B 0.000,C 90.000,E1 47.067} C_DIS
LIN {X 0.146,Y -223.657,Z 1896.245,A 0.000,B 0.000,C 90.000,E1 44.028} C_DIS
LIN {X -0.116,Y -212.645,Z 1896.225,A 0.000,B 0.000,C 90.000,E1 40.620} C_DIS
LIN {X -0.043,Y -203.662,Z 1896.208,A 0.000,B 0.000,C 90.000,E1 37.443} C_DIS
LIN {X 0.071,Y -195.559,Z 1896.190,A 0.000,B 0.000,C 90.000,E1 34.199} C_DIS
LIN {X 0.086,Y -188.184,Z 1896.172,A 0.000,B 0.000,C 90.000,E1 30.924} C_DIS
LIN {X -0.042,Y -181.537,Z 1896.153,A 0.000,B 0.000,C 90.000,E1 27.641} C_DIS
LIN {X -0.012,Y -175.602,Z 1896.135,A 0.000,B 0.000,C 90.000,E1 24.259} C_DIS
LIN {X -0.022,Y -170.497,Z 1896.116,A 0.000,B 0.000,C 90.000,E1 20.844} C_DIS
LIN {X -0.071,Y -166.189,Z 1896.097,A 0.000,B 0.000,C 90.000,E1 17.402} C_DIS
LIN {X 0.001,Y -162.661,Z 1896.077,A 0.000,B 0.000,C 90.000,E1 13.883} C_DIS
LIN {X -0.014,Y -159.714,Z 1896.058,A 0.000,B 0.000,C 90.000,E1 10.366} C_DIS
LIN {X 0.039,Y -157.117,Z 1896.033,A 0.000,B 0.000,C 90.000,E1 5.910} C_DIS
LIN {X 0.000,Y -154.868,Z 1896.000,A 0.000,B 0.000,C 90.000,E1 360.000} C_DIS
LIN {X -0.013,Y -154.104,Z 1895.948,A 0.000,B 0.000,C 90.000,E1 350.557} C_DIS
LIN {X -0.010,Y -156.115,Z 1895.908,A 0.000,B 0.000,C 90.000,E1 343.378} C_DIS
LIN {X 0.023,Y -158.532,Z 1895.883,A 0.000,B 0.000,C 90.000,E1 338.901} C_DIS
LIN {X 0.036,Y -162.146,Z 1895.858,A 0.000,B 0.000,C 90.000,E1 334.460} C_DIS
LIN {X 0.087,Y -166.099,Z 1895.839,A 0.000,B 0.000,C 90.000,E1 330.923} C_DIS
LIN {X 0.020,Y -169.692,Z 1895.824,A 0.000,B 0.000,C 90.000,E1 328.329} C_DIS
LIN {X 0.055,Y -173.830,Z 1895.810,A 0.000,B 0.000,C 90.000,E1 325.722} C_DIS
LIN {X -0.021,Y -178.581,Z 1895.795,A 0.000,B 0.000,C 90.000,E1 323.176} C_DIS
LIN {X -0.049,Y -184.145,Z 1895.781,A 0.000,B 0.000,C 90.000,E1 320.642} C_DIS
LIN {X 0.005,Y -190.612,Z 1895.767,A 0.000,B 0.000,C 90.000,E1 318.119} C_DIS
LIN {X 0.019,Y -198.093,Z 1895.754,A 0.000,B 0.000,C 90.000,E1 315.648} C_DIS
LIN {X 0.039,Y -206.519,Z 1895.740,A 0.000,B 0.000,C 90.000,E1 313.218} C_DIS
LIN {X -0.006,Y -217.469,Z 1895.725,A 0.000,B 0.000,C 90.000,E1 310.458} C_DIS
LIN {X 0.024,Y -231.231,Z 1895.708,A 0.000,B 0.000,C 90.000,E1 307.363} C_DIS
LIN {X -0.155,Y -246.185,Z 1895.691,A 0.000,B 0.000,C 90.000,E1 304.405} C_DIS
LIN {X -0.149,Y -258.035,Z 1895.679,A 0.000,B 0.000,C 90.000,E1 302.212} C_DIS
LIN {X 0.095,Y -272.095,Z 1895.665,A 0.000,B 0.000,C 90.000,E1 299.667} C_DIS
LIN {X -0.129,Y -281.986,Z 1895.655,A 0.000,B 0.000,C 90.000,E1 297.975} C_DIS
LIN {X 0.026,Y -285.864,Z 1895.651,A 0.000,B 0.000,C 90.000,E1 297.257} C_DIS
LIN {X -0.058,Y -295.849,Z 1895.643,A 0.000,B 0.000,C 90.000,E1 295.771} C_DIS
LIN {X -0.016,Y -308.956,Z 1895.632,A 0.000,B 0.000,C 90.000,E1 293.770} C_DIS
LIN {X -0.052,Y -319.583,Z 1895.623,A 0.000,B 0.000,C 90.000,E1 292.153} C_DIS
LIN {X 0.001,Y -327.767,Z 1895.616,A 0.000,B 0.000,C 90.000,E1 290.865} C_DIS
LIN {X -0.153,Y -335.501,Z 1895.609,A 0.000,B 0.000,C 90.000,E1 289.631} C_DIS
LIN {X -0.011,Y -342.760,Z 1895.602,A 0.000,B 0.000,C 90.000,E1 288.362} C_DIS
LIN {X -0.117,Y -347.719,Z 1895.597,A 0.000,B 0.000,C 90.000,E1 287.457} C_DIS
LIN {X 0.162,Y -352.078,Z 1895.592,A 0.000,B 0.000,C 90.000,E1 286.496} C_DIS
LIN {X 0.044,Y -355.835,Z 1895.587,A 0.000,B 0.000,C 90.000,E1 285.607} C_DIS
LIN {X 0.017,Y -358.046,Z 1895.583,A 0.000,B 0.000,C 90.000,E1 285.009} C_DIS
LIN {X 0.003,Y -360.007,Z 1895.580,A 0.000,B 0.000,C 90.000,E1 284.411} C_DIS
LIN {X -0.096,Y -361.662,Z 1895.577,A 0.000,B 0.000,C 90.000,E1 283.828} C_DIS
LIN {X -0.096,Y -362.987,Z 1895.573,A 0.000,B 0.000,C 90.000,E1 283.231} C_DIS
LIN {X 0.186,Y -363.967,Z 1895.570,A 0.000,B 0.000,C 90.000,E1 282.591} C_DIS
LIN {X 0.122,Y -364.489,Z 1895.567,A 0.000,B 0.000,C 90.000,E1 282.007} C_DIS
LIN {X 0.066,Y -364.682,Z 1895.563,A 0.000,B 0.000,C 90.000,E1 281.422} C_DIS
LIN {X 0.013,Y -364.441,Z 1895.560,A 0.000,B 0.000,C 90.000,E1 280.838} C_DIS
LIN {X -0.039,Y -363.851,Z 1895.557,A 0.000,B 0.000,C 90.000,E1 280.254} C_DIS
LIN {X -0.094,Y -362.857,Z 1895.554,A 0.000,B 0.000,C 90.000,E1 279.670} C_DIS
LIN {X 0.203,Y -361.491,Z 1895.550,A 0.000,B 0.000,C 90.000,E1 279.029} C_DIS
LIN {X 0.080,Y -359.788,Z 1895.547,A 0.000,B 0.000,C 90.000,E1 278.454} C_DIS
LIN {X -0.089,Y -356.702,Z 1895.542,A 0.000,B 0.000,C 90.000,E1 277.587} C_DIS
LIN {X 0.164,Y -354.198,Z 1895.539,A 0.000,B 0.000,C 90.000,E1 276.947} C_DIS
LIN {X 0.004,Y -351.255,Z 1895.535,A 0.000,B 0.000,C 90.000,E1 276.372} C_DIS
LIN {X 0.069,Y -345.935,Z 1895.530,A 0.000,B 0.000,C 90.000,E1 275.454} C_DIS
LIN {X -0.129,Y -341.597,Z 1895.527,A 0.000,B 0.000,C 90.000,E1 274.878} C_DIS
LIN {X -0.010,Y -336.714,Z 1895.524,A 0.000,B 0.000,C 90.000,E1 274.245} C_DIS
LIN {X 0.076,Y -331.094,Z 1895.520,A 0.000,B 0.000,C 90.000,E1 273.612} C_DIS
LIN {X 0.045,Y -325.005,Z 1895.517,A 0.000,B 0.000,C 90.000,E1 273.037} C_DIS
LIN {X 0.001,Y -318.767,Z 1895.514,A 0.000,B 0.000,C 90.000,E1 272.522} C_DIS
LIN {X -0.059,Y -312.426,Z 1895.511,A 0.000,B 0.000,C 90.000,E1 272.064} C_DIS
LIN {X 0.141,Y -305.464,Z 1895.509,A 0.000,B 0.000,C 90.000,E1 271.604} C_DIS
LIN {X 0.056,Y -298.315,Z 1895.507,A 0.000,B 0.000,C 90.000,E1 271.260} C_DIS
LIN {X 0.000,Y -290.641,Z 1895.505,A 0.000,B 0.000,C 90.000,E1 270.974} C_DIS
LIN {X 0.011,Y -282.405,Z 1895.504,A 0.000,B 0.000,C 90.000,E1 270.745} C_DIS
LIN {X 0.043,Y -274.132,Z 1895.503,A 0.000,B 0.000,C 90.000,E1 270.573} C_DIS
LIN {X -0.001,Y -260.348,Z 1895.502,A 0.000,B 0.000,C 90.000,E1 270.401} C_DIS
LIN {X 0.119,Y -246.916,Z 1895.502,A 0.000,B 0.000,C 90.000,E1 270.286} C_DIS
LIN {X 0.062,Y -181.581,Z 1895.502,A 0.000,B 0.000,C 90.000,E1 270.286} C_DIS
LIN {X 0.024,Y -180.837,Z 1895.472,A 0.000,B 0.000,C 90.000,E1 264.894} C_DIS
LIN {X -0.073,Y -178.943,Z 1895.443,A 0.000,B 0.000,C 90.000,E1 259.859} C_DIS
LIN {X -0.029,Y -175.995,Z 1895.415,A 0.000,B 0.000,C 90.000,E1 254.755} C_DIS
LIN {X -0.083,Y -175.500,Z 1895.411,A 0.000,B 0.000,C 90.000,E1 253.921} C_DIS
LIN {X -0.020,Y -172.241,Z 1895.387,A 0.000,B 0.000,C 90.000,E1 249.625} C_DIS
LIN {X -0.041,Y -171.719,Z 1895.382,A 0.000,B 0.000,C 90.000,E1 248.773} C_DIS
LIN {X -0.032,Y -167.315,Z 1895.353,A 0.000,B 0.000,C 90.000,E1 243.589} C_DIS
LIN {X 0.049,Y -166.696,Z 1895.348,A 0.000,B 0.000,C 90.000,E1 242.692} C_DIS
LIN {X 0.039,Y -162.677,Z 1895.324,A 0.000,B 0.000,C 90.000,E1 238.329} C_DIS
LIN {X 0.011,Y -161.367,Z 1895.314,A 0.000,B 0.000,C 90.000,E1 236.580} C_DIS
LIN {X -0.079,Y -157.361,Z 1895.290,A 0.000,B 0.000,C 90.000,E1 232.190} C_DIS
LIN {X 0.073,Y -155.350,Z 1895.275,A 0.000,B 0.000,C 90.000,E1 229.461} C_DIS
LIN {X 0.003,Y -151.696,Z 1895.250,A 0.000,B 0.000,C 90.000,E1 225.000} C_DIS
LIN {X 0.051,Y -150.558,Z 1895.240,A 0.000,B 0.000,C 90.000,E1 223.176} C_DIS
LIN {X -0.032,Y -147.284,Z 1895.215,A 0.000,B 0.000,C 90.000,E1 218.669} C_DIS
LIN {X -0.063,Y -145.313,Z 1895.194,A 0.000,B 0.000,C 90.000,E1 215.025} C_DIS
LIN {X 0.047,Y -142.402,Z 1895.164,A 0.000,B 0.000,C 90.000,E1 209.461} C_DIS
LIN {X 0.029,Y -141.384,Z 1895.148,A 0.000,B 0.000,C 90.000,E1 206.693} C_DIS
LIN {X 0.022,Y -139.350,Z 1895.112,A 0.000,B 0.000,C 90.000,E1 200.194} C_DIS
LIN {X 0.012,Y -138.788,Z 1895.097,A 0.000,B 0.000,C 90.000,E1 197.402} C_DIS
LIN {X -0.066,Y -138.344,Z 1895.055,A 0.000,B 0.000,C 90.000,E1 189.962} C_DIS
LIN {X -0.048,Y -139.384,Z 1895.008,A 0.000,B 0.000,C 90.000,E1 181.547} C_DIS
LIN {X 0.005,Y -141.280,Z 1894.972,A 0.000,B 0.000,C 90.000,E1 175.008} C_DIS
LIN {X -0.037,Y -142.644,Z 1894.957,A 0.000,B 0.000,C 90.000,E1 172.243} C_DIS
LIN {X 0.055,Y -144.979,Z 1894.931,A 0.000,B 0.000,C 90.000,E1 167.589} C_DIS
LIN {X 0.045,Y -147.606,Z 1894.911,A 0.000,B 0.000,C 90.000,E1 163.921} C_DIS
LIN {X -0.017,Y -150.227,Z 1894.891,A 0.000,B 0.000,C 90.000,E1 160.296} C_DIS
LIN {X -0.001,Y -153.618,Z 1894.870,A 0.000,B 0.000,C 90.000,E1 156.666} C_DIS
LIN {X -0.014,Y -157.033,Z 1894.850,A 0.000,B 0.000,C 90.000,E1 153.076} C_DIS
LIN {X -0.083,Y -161.157,Z 1894.831,A 0.000,B 0.000,C 90.000,E1 149.537} C_DIS
LIN {X 0.000,Y -163.254,Z 1894.821,A 0.000,B 0.000,C 90.000,E1 147.740} C_DIS
LIN {X 0.099,Y -167.691,Z 1894.801,A 0.000,B 0.000,C 90.000,E1 144.196} C_DIS
LIN {X 0.012,Y -171.513,Z 1894.787,A 0.000,B 0.000,C 90.000,E1 141.618} C_DIS
LIN {X 0.056,Y -176.449,Z 1894.768,A 0.000,B 0.000,C 90.000,E1 138.162} C_DIS
LIN {X -0.074,Y -180.746,Z 1894.753,A 0.000,B 0.000,C 90.000,E1 135.648} C_DIS
LIN {X 0.044,Y -186.151,Z 1894.735,A 0.000,B 0.000,C 90.000,E1 132.243} C_DIS
LIN {X -0.037,Y -190.788,Z 1894.721,A 0.000,B 0.000,C 90.000,E1 129.769} C_DIS
LIN {X 0.028,Y -196.544,Z 1894.703,A 0.000,B 0.000,C 90.000,E1 126.457} C_DIS
LIN {X -0.053,Y -201.317,Z 1894.689,A 0.000,B 0.000,C 90.000,E1 124.040} C_DIS
LIN {X 0.043,Y -207.288,Z 1894.671,A 0.000,B 0.000,C 90.000,E1 120.797} C_DIS
LIN {X 0.043,Y -210.542,Z 1894.662,A 0.000,B 0.000,C 90.000,E1 119.205} C_DIS
LIN {X 0.045,Y -216.347,Z 1894.645,A 0.000,B 0.000,C 90.000,E1 116.052} C_DIS
LIN {X -0.047,Y -219.484,Z 1894.636,A 0.000,B 0.000,C 90.000,E1 114.515} C_DIS
LIN {X -0.047,Y -224.133,Z 1894.621,A 0.000,B 0.000,C 90.000,E1 111.844} C_DIS
LIN {X -0.094,Y -283.790,Z 1894.621,A 0.000,B 0.000,C 90.000,E1 111.844} C_DIS
LIN {X 0.053,Y -286.026,Z 1894.621,A 0.000,B 0.000,C 90.000,E1 111.770} C_DIS
LIN {X 0.031,Y -289.714,Z 1894.620,A 0.000,B 0.000,C 90.000,E1 111.589} C_DIS
LIN {X 0.009,Y -291.934,Z 1894.619,A 0.000,B 0.000,C 90.000,E1 111.408} C_DIS
LIN {X -0.004,Y -295.808,Z 1894.616,A 0.000,B 0.000,C 90.000,E1 110.918} C_DIS
LIN {X 0.164,Y -311.070,Z 1894.601,A 0.000,B 0.000,C 90.000,E1 108.236} C_DIS
LIN {X -0.091,Y -325.816,Z 1894.589,A 0.000,B 0.000,C 90.000,E1 106.024} C_DIS
LIN {X -0.006,Y -339.654,Z 1894.578,A 0.000,B 0.000,C 90.000,E1 104.120} C_DIS
LIN {X -0.149,Y -354.680,Z 1894.568,A 0.000,B 0.000,C 90.000,E1 102.299} C_DIS
LIN {X 0.000,Y -373.156,Z 1894.557,A 0.000,B 0.000,C 90.000,E1 100.254} C_DIS
LIN {X 0.158,Y -392.028,Z 1894.547,A 0.000,B 0.000,C 90.000,E1 98.398} C_DIS
LIN {X -0.206,Y -411.309,Z 1894.537,A 0.000,B 0.000,C 90.000,E1 96.777} C_DIS
LIN {X 0.174,Y -433.722,Z 1894.528,A 0.000,B 0.000,C 90.000,E1 94.992} C_DIS
LIN {X 0.160,Y -439.358,Z 1894.526,A 0.000,B 0.000,C 90.000,E1 94.588} C_DIS
LIN {X 0.136,Y -443.342,Z 1894.523,A 0.000,B 0.000,C 90.000,E1 94.188} C_DIS
LIN {X -0.040,Y -445.040,Z 1894.522,A 0.000,B 0.000,C 90.000,E1 93.955} C_DIS
LIN {X 0.196,Y -446.334,Z 1894.521,A 0.000,B 0.000,C 90.000,E1 93.669} C_DIS
LIN {X 0.122,Y -448.039,Z 1894.518,A 0.000,B 0.000,C 90.000,E1 93.154} C_DIS
LIN {X 0.080,Y -448.705,Z 1894.515,A 0.000,B 0.000,C 90.000,E1 92.636} C_DIS
LIN {X 0.026,Y -448.439,Z 1894.512,A 0.000,B 0.000,C 90.000,E1 92.121} C_DIS
LIN {X -0.009,Y -447.208,Z 1894.509,A 0.000,B 0.000,C 90.000,E1 91.604} C_DIS
LIN {X 0.189,Y -446.174,Z 1894.507,A 0.000,B 0.000,C 90.000,E1 91.318} C_DIS
LIN {X -0.060,Y -444.797,Z 1894.506,A 0.000,B 0.000,C 90.000,E1 91.088} C_DIS
LIN {X 0.025,Y -431.638,Z 1894.494,A 0.000,B 0.000,C 90.000,E1 88.969} C_DIS
LIN {X 0.004,Y -421.572,Z 1894.485,A 0.000,B 0.000,C 90.000,E1 87.364} C_DIS
LIN {X -0.086,Y -409.791,Z 1894.475,A 0.000,B 0.000,C 90.000,E1 85.469} C_DIS
LIN {X 0.021,Y -397.903,Z 1894.464,A 0.000,B 0.000,C 90.000,E1 83.514} C_DIS
LIN {X -0.032,Y -385.931,Z 1894.453,A 0.000,B 0.000,C 90.000,E1 81.546} C_DIS
LIN {X 0.115,Y -374.072,Z 1894.442,A 0.000,B 0.000,C 90.000,E1 79.511} C_DIS
LIN {X 0.023,Y -356.041,Z 1894.424,A 0.000,B 0.000,C 90.000,E1 76.284} C_DIS
LIN {X 0.044,Y -342.233,Z 1894.409,A 0.000,B 0.000,C 90.000,E1 73.559} C_DIS
LIN {X 0.002,Y -330.355,Z 1894.395,A 0.000,B 0.000,C 90.000,E1 71.094} C_DIS
LIN {X 0.124,Y -317.320,Z 1894.379,A 0.000,B 0.000,C 90.000,E1 68.230} C_DIS
LIN {X -0.047,Y -304.920,Z 1894.363,A 0.000,B 0.000,C 90.000,E1 65.357} C_DIS
LIN {X -0.035,Y -295.396,Z 1894.350,A 0.000,B 0.000,C 90.000,E1 63.050} C_DIS
LIN {X -0.086,Y -286.084,Z 1894.337,A 0.000,B 0.000,C 90.000,E1 60.717} C_DIS
LIN {X -0.067,Y -276.648,Z 1894.324,A 0.000,B 0.000,C 90.000,E1 58.329} C_DIS
LIN {X 0.033,Y -267.162,Z 1894.311,A 0.000,B 0.000,C 90.000,E1 55.881} C_DIS
LIN {X -0.004,Y -257.541,Z 1894.297,A 0.000,B 0.000,C 90.000,E1 53.417} C_DIS
LIN {X 0.060,Y -247.946,Z 1894.283,A 0.000,B 0.000,C 90.000,E1 50.884} C_DIS
LIN {X 0.012,Y -237.102,Z 1894.266,A 0.000,B 0.000,C 90.000,E1 47.957} C_DIS
LIN {X -0.067,Y -225.366,Z 1894.248,A 0.000,B 0.000,C 90.000,E1 44.595} C_DIS
LIN {X -0.046,Y -215.410,Z 1894.231,A 0.000,B 0.000,C 90.000,E1 41.515} C_DIS
LIN {X -0.071,Y -206.185,Z 1894.213,A 0.000,B 0.000,C 90.000,E1 38.382} C_DIS
LIN {X -0.100,Y -198.855,Z 1894.198,A 0.000,B 0.000,C 90.000,E1 35.598} C_DIS
LIN {X -0.053,Y -191.184,Z 1894.180,A 0.000,B 0.000,C 90.000,E1 32.339} C_DIS
LIN {X -0.012,Y -184.240,Z 1894.161,A 0.000,B 0.000,C 90.000,E1 29.027} C_DIS
LIN {X 0.009,Y -177.976,Z 1894.143,A 0.000,B 0.000,C 90.000,E1 25.668} C_DIS
LIN {X -0.019,Y -173.825,Z 1894.128,A 0.000,B 0.000,C 90.000,E1 23.131} C_DIS
LIN {X 0.022,Y -168.958,Z 1894.109,A 0.000,B 0.000,C 90.000,E1 19.685} C_DIS
LIN {X 0.045,Y -164.939,Z 1894.090,A 0.000,B 0.000,C 90.000,E1 16.205} C_DIS
LIN {X 0.027,Y -160.868,Z 1894.066,A 0.000,B 0.000,C 90.000,E1 11.827} C_DIS
LIN {X 0.064,Y -158.349,Z 1894.046,A 0.000,B 0.000,C 90.000,E1 8.276} C_DIS
LIN {X -0.005,Y -155.523,Z 1894.011,A 0.000,B 0.000,C 90.000,E1 2.064} C_DIS
LIN {X 0.048,Y -154.021,Z 1893.953,A 0.000,B 0.000,C 90.000,E1 351.432} C_DIS
LIN {X -0.038,Y -155.760,Z 1893.913,A 0.000,B 0.000,C 90.000,E1 344.283} C_DIS
LIN {X 0.022,Y -158.529,Z 1893.883,A 0.000,B 0.000,C 90.000,E1 338.901} C_DIS
LIN {X 0.035,Y -162.145,Z 1893.858,A 0.000,B 0.000,C 90.000,E1 334.460} C_DIS
LIN {X 0.087,Y -166.102,Z 1893.839,A 0.000,B 0.000,C 90.000,E1 330.923} C_DIS
LIN {X 0.019,Y -169.696,Z 1893.824,A 0.000,B 0.000,C 90.000,E1 328.329} C_DIS
LIN {X 0.054,Y -173.837,Z 1893.810,A 0.000,B 0.000,C 90.000,E1 325.722} C_DIS
LIN {X -0.022,Y -178.588,Z 1893.795,A 0.000,B 0.000,C 90.000,E1 323.176} C_DIS
LIN {X -0.050,Y -184.154,Z 1893.781,A 0.000,B 0.000,C 90.000,E1 320.642} C_DIS
LIN {X 0.004,Y -190.621,Z 1893.767,A 0.000,B 0.000,C 90.000,E1 318.119} C_DIS
LIN {X 0.018,Y -198.099,Z 1893.754,A 0.000,B 0.000,C 90.000,E1 315.648} C_DIS
LIN {X 0.039,Y -206.524,Z 1893.740,A 0.000,B 0.000,C 90.000,E1 313.218} C_DIS
LIN {X -0.006,Y -217.477,Z 1893.725,A 0.000,B 0.000,C 90.000,E1 310.458} C_DIS
LIN {X 0.079,Y -229.448,Z 1893.710,A 0.000,B 0.000,C 90.000,E1 307.729} C_DIS
LIN {X -0.002,Y -244.277,Z 1893.693,A 0.000,B 0.000,C 90.000,E1 304.739} C_DIS
LIN {X -0.149,Y -258.044,Z 1893.679,A 0.000,B 0.000,C 90.000,E1 302.212} C_DIS
LIN {X 0.096,Y -272.102,Z 1893.665,A 0.000,B 0.000,C 90.000,E1 299.667} C_DIS
LIN {X -0.128,Y -281.995,Z 1893.655,A 0.000,B 0.000,C 90.000,E1 297.975} C_DIS
LIN {X -0.047,Y -292.097,Z 1893.647,A 0.000,B 0.000,C 90.000,E1 296.411} C_DIS
LIN {X 0.050,Y -305.304,Z 1893.635,A 0.000,B 0.000,C 90.000,E1 294.387} C_DIS
LIN {X -0.045,Y -316.100,Z 1893.626,A 0.000,B 0.000,C 90.000,E1 292.770} C_DIS
LIN {X 0.020,Y -326.538,Z 1893.618,A 0.000,B 0.000,C 90.000,E1 291.153} C_DIS
LIN {X 0.047,Y -334.386,Z 1893.610,A 0.000,B 0.000,C 90.000,E1 289.885} C_DIS
LIN {X -0.032,Y -341.801,Z 1893.604,A 0.000,B 0.000,C 90.000,E1 288.652} C_DIS
LIN {X 0.186,Y -346.917,Z 1893.599,A 0.000,B 0.000,C 90.000,E1 287.692} C_DIS
LIN {X 0.017,Y -351.456,Z 1893.593,A 0.000,B 0.000,C 90.000,E1 286.804} C_DIS
LIN {X -0.005,Y -355.363,Z 1893.588,A 0.000,B 0.000,C 90.000,E1 285.898} C_DIS
LIN {X -0.096,Y -358.752,Z 1893.583,A 0.000,B 0.000,C 90.000,E1 285.009} C_DIS
LIN {X -0.107,Y -360.685,Z 1893.580,A 0.000,B 0.000,C 90.000,E1 284.411} C_DIS
LIN {X 0.151,Y -362.329,Z 1893.577,A 0.000,B 0.000,C 90.000,E1 283.772} C_DIS
LIN {X 0.156,Y -363.623,Z 1893.573,A 0.000,B 0.000,C 90.000,E1 283.175} C_DIS
LIN {X 0.088,Y -364.528,Z 1893.570,A 0.000,B 0.000,C 90.000,E1 282.591} C_DIS
LIN {X 0.028,Y -365.051,Z 1893.567,A 0.000,B 0.000,C 90.000,E1 282.007} C_DIS
LIN {X -0.024,Y -365.165,Z 1893.563,A 0.000,B 0.000,C 90.000,E1 281.422} C_DIS
LIN {X -0.074,Y -364.906,Z 1893.560,A 0.000,B 0.000,C 90.000,E1 280.838} C_DIS
LIN {X -0.123,Y -364.298,Z 1893.557,A 0.000,B 0.000,C 90.000,E1 280.254} C_DIS
LIN {X 0.183,Y -363.280,Z 1893.554,A 0.000,B 0.000,C 90.000,E1 279.613} C_DIS
LIN {X 0.125,Y -361.885,Z 1893.550,A 0.000,B 0.000,C 90.000,E1 279.029} C_DIS
LIN {X 0.006,Y -360.157,Z 1893.547,A 0.000,B 0.000,C 90.000,E1 278.454} C_DIS
LIN {X -0.159,Y -357.017,Z 1893.542,A 0.000,B 0.000,C 90.000,E1 277.587} C_DIS
LIN {X 0.000,Y -353.050,Z 1893.537,A 0.000,B 0.000,C 90.000,E1 276.663} C_DIS
LIN {X 0.114,Y -348.060,Z 1893.532,A 0.000,B 0.000,C 90.000,E1 275.739} C_DIS
LIN {X -0.076,Y -344.039,Z 1893.529,A 0.000,B 0.000,C 90.000,E1 275.163} C_DIS
LIN {X 0.054,Y -339.402,Z 1893.525,A 0.000,B 0.000,C 90.000,E1 274.531} C_DIS
LIN {X 0.154,Y -334.081,Z 1893.522,A 0.000,B 0.000,C 90.000,E1 273.898} C_DIS
LIN {X -0.007,Y -328.263,Z 1893.518,A 0.000,B 0.000,C 90.000,E1 273.326} C_DIS
LIN {X 0.136,Y -322.130,Z 1893.515,A 0.000,B 0.000,C 90.000,E1 272.751} C_DIS
LIN {X -0.036,Y -315.903,Z 1893.513,A 0.000,B 0.000,C 90.000,E1 272.293} C_DIS
LIN {X 0.073,Y -309.332,Z 1893.510,A 0.000,B 0.000,C 90.000,E1 271.835} C_DIS
LIN {X 0.143,Y -302.364,Z 1893.508,A 0.000,B 0.000,C 90.000,E1 271.432} C_DIS
LIN {X -0.077,Y -295.076,Z 1893.506,A 0.000,B 0.000,C 90.000,E1 271.146} C_DIS
LIN {X 0.052,Y -287.288,Z 1893.505,A 0.000,B 0.000,C 90.000,E1 270.859} C_DIS
LIN {X 0.056,Y -275.628,Z 1893.503,A 0.000,B 0.000,C 90.000,E1 270.573} C_DIS
LIN {X 0.103,Y -263.339,Z 1893.502,A 0.000,B 0.000,C 90.000,E1 270.344} C_DIS
LIN {X 0.095,Y -249.152,Z 1893.501,A 0.000,B 0.000,C 90.000,E1 270.172} C_DIS
LIN {X -0.114,Y -240.995,Z 1893.501,A 0.000,B 0.000,C 90.000,E1 270.172} C_DIS
LIN {X 0.065,Y -181.576,Z 1893.501,A 0.000,B 0.000,C 90.000,E1 270.115} C_DIS
LIN {X -0.044,Y -180.908,Z 1893.475,A 0.000,B 0.000,C 90.000,E1 265.584} C_DIS
LIN {X 0.014,Y -180.778,Z 1893.471,A 0.000,B 0.000,C 90.000,E1 264.723} C_DIS
LIN {X -0.092,Y -178.875,Z 1893.443,A 0.000,B 0.000,C 90.000,E1 259.690} C_DIS
LIN {X -0.016,Y -175.917,Z 1893.414,A 0.000,B 0.000,C 90.000,E1 254.574} C_DIS
LIN {X 0.040,Y -174.611,Z 1893.405,A 0.000,B 0.000,C 90.000,E1 252.851} C_DIS
LIN {X -0.033,Y -171.592,Z 1893.381,A 0.000,B 0.000,C 90.000,E1 248.592} C_DIS
LIN {X -0.044,Y -167.814,Z 1893.357,A 0.000,B 0.000,C 90.000,E1 244.280} C_DIS
LIN {X -0.026,Y -166.536,Z 1893.347,A 0.000,B 0.000,C 90.000,E1 242.538} C_DIS
LIN {X 0.023,Y -162.535,Z 1893.323,A 0.000,B 0.000,C 90.000,E1 238.152} C_DIS
LIN {X -0.055,Y -161.210,Z 1893.313,A 0.000,B 0.000,C 90.000,E1 236.421} C_DIS
LIN {X -0.019,Y -157.218,Z 1893.289,A 0.000,B 0.000,C 90.000,E1 231.984} C_DIS
LIN {X 0.004,Y -155.945,Z 1893.279,A 0.000,B 0.000,C 90.000,E1 230.194} C_DIS
LIN {X -0.037,Y -152.197,Z 1893.254,A 0.000,B 0.000,C 90.000,E1 225.729} C_DIS
LIN {X -0.016,Y -150.443,Z 1893.239,A 0.000,B 0.000,C 90.000,E1 223.014} C_DIS
LIN {X 0.012,Y -147.170,Z 1893.214,A 0.000,B 0.000,C 90.000,E1 218.463} C_DIS
LIN {X -0.022,Y -145.186,Z 1893.193,A 0.000,B 0.000,C 90.000,E1 214.818} C_DIS
LIN {X 0.014,Y -142.329,Z 1893.163,A 0.000,B 0.000,C 90.000,E1 209.283} C_DIS
LIN {X 0.009,Y -141.718,Z 1893.152,A 0.000,B 0.000,C 90.000,E1 207.436} C_DIS
LIN {X 0.056,Y -139.476,Z 1893.116,A 0.000,B 0.000,C 90.000,E1 200.918} C_DIS
LIN {X 0.047,Y -138.973,Z 1893.101,A 0.000,B 0.000,C 90.000,E1 198.127} C_DIS
LIN {X 0.036,Y -138.330,Z 1893.054,A 0.000,B 0.000,C 90.000,E1 189.726} C_DIS
LIN {X 0.039,Y -139.435,Z 1893.007,A 0.000,B 0.000,C 90.000,E1 181.318} C_DIS
LIN {X -0.021,Y -140.963,Z 1892.976,A 0.000,B 0.000,C 90.000,E1 175.755} C_DIS
LIN {X 0.070,Y -142.719,Z 1892.956,A 0.000,B 0.000,C 90.000,E1 172.008} C_DIS
LIN {X 0.028,Y -145.099,Z 1892.930,A 0.000,B 0.000,C 90.000,E1 167.409} C_DIS
LIN {X 0.023,Y -147.723,Z 1892.910,A 0.000,B 0.000,C 90.000,E1 163.740} C_DIS
LIN {X -0.036,Y -150.384,Z 1892.889,A 0.000,B 0.000,C 90.000,E1 160.115} C_DIS
LIN {X -0.018,Y -153.815,Z 1892.869,A 0.000,B 0.000,C 90.000,E1 156.485} C_DIS
LIN {X 0.041,Y -157.227,Z 1892.849,A 0.000,B 0.000,C 90.000,E1 152.871} C_DIS
LIN {X -0.018,Y -161.394,Z 1892.830,A 0.000,B 0.000,C 90.000,E1 149.331} C_DIS
LIN {X -0.008,Y -165.596,Z 1892.810,A 0.000,B 0.000,C 90.000,E1 145.801} C_DIS
LIN {X -0.022,Y -170.520,Z 1892.791,A 0.000,B 0.000,C 90.000,E1 142.316} C_DIS
LIN {X 0.022,Y -175.400,Z 1892.771,A 0.000,B 0.000,C 90.000,E1 138.852} C_DIS
LIN {X 0.013,Y -181.023,Z 1892.752,A 0.000,B 0.000,C 90.000,E1 135.445} C_DIS
LIN {X 0.007,Y -186.455,Z 1892.734,A 0.000,B 0.000,C 90.000,E1 132.081} C_DIS
LIN {X 0.076,Y -191.079,Z 1892.720,A 0.000,B 0.000,C 90.000,E1 129.564} C_DIS
LIN {X -0.002,Y -196.868,Z 1892.702,A 0.000,B 0.000,C 90.000,E1 126.297} C_DIS
LIN {X -0.085,Y -200.127,Z 1892.693,A 0.000,B 0.000,C 90.000,E1 124.692} C_DIS
LIN {X -0.093,Y -207.623,Z 1892.670,A 0.000,B 0.000,C 90.000,E1 120.669} C_DIS
LIN {X -0.091,Y -210.821,Z 1892.661,A 0.000,B 0.000,C 90.000,E1 119.077} C_DIS
LIN {X 0.010,Y -216.672,Z 1892.644,A 0.000,B 0.000,C 90.000,E1 115.899} C_DIS
LIN {X 0.026,Y -219.746,Z 1892.635,A 0.000,B 0.000,C 90.000,E1 114.335} C_DIS
LIN {X -0.027,Y -224.123,Z 1892.621,A 0.000,B 0.000,C 90.000,E1 111.844} C_DIS
LIN {X -0.068,Y -283.137,Z 1892.621,A 0.000,B 0.000,C 90.000,E1 111.844} C_DIS
LIN {X 0.016,Y -286.298,Z 1892.621,A 0.000,B 0.000,C 90.000,E1 111.770} C_DIS
LIN {X -0.122,Y -290.813,Z 1892.620,A 0.000,B 0.000,C 90.000,E1 111.535} C_DIS
LIN {X 0.120,Y -293.415,Z 1892.618,A 0.000,B 0.000,C 90.000,E1 111.227} C_DIS
LIN {X 0.080,Y -297.163,Z 1892.615,A 0.000,B 0.000,C 90.000,E1 110.663} C_DIS
LIN {X -0.011,Y -310.489,Z 1892.602,A 0.000,B 0.000,C 90.000,E1 108.362} C_DIS
LIN {X 0.114,Y -325.184,Z 1892.589,A 0.000,B 0.000,C 90.000,E1 106.079} C_DIS
LIN {X 0.109,Y -338.967,Z 1892.579,A 0.000,B 0.000,C 90.000,E1 104.189} C_DIS
LIN {X 0.035,Y -353.943,Z 1892.569,A 0.000,B 0.000,C 90.000,E1 102.355} C_DIS
LIN {X 0.163,Y -372.363,Z 1892.557,A 0.000,B 0.000,C 90.000,E1 100.310} C_DIS
LIN {X -0.134,Y -391.257,Z 1892.547,A 0.000,B 0.000,C 90.000,E1 98.511} C_DIS
LIN {X -0.131,Y -410.491,Z 1892.538,A 0.000,B 0.000,C 90.000,E1 96.834} C_DIS
LIN {X 0.201,Y -432.887,Z 1892.528,A 0.000,B 0.000,C 90.000,E1 95.049} C_DIS
LIN {X 0.177,Y -438.544,Z 1892.526,A 0.000,B 0.000,C 90.000,E1 94.645} C_DIS
LIN {X -0.054,Y -441.008,Z 1892.525,A 0.000,B 0.000,C 90.000,E1 94.473} C_DIS
LIN {X 0.086,Y -444.590,Z 1892.522,A 0.000,B 0.000,C 90.000,E1 94.012} C_DIS
LIN {X -0.187,Y -446.027,Z 1892.521,A 0.000,B 0.000,C 90.000,E1 93.784} C_DIS
LIN {X -0.015,Y -447.105,Z 1892.519,A 0.000,B 0.000,C 90.000,E1 93.498} C_DIS
LIN {X -0.059,Y -448.390,Z 1892.516,A 0.000,B 0.000,C 90.000,E1 92.980} C_DIS
LIN {X -0.121,Y -448.698,Z 1892.514,A 0.000,B 0.000,C 90.000,E1 92.465} C_DIS
LIN {X -0.171,Y -448.078,Z 1892.511,A 0.000,B 0.000,C 90.000,E1 91.949} C_DIS
LIN {X -0.207,Y -446.439,Z 1892.508,A 0.000,B 0.000,C 90.000,E1 91.432} C_DIS
LIN {X -0.009,Y -445.151,Z 1892.506,A 0.000,B 0.000,C 90.000,E1 91.146} C_DIS
LIN {X -0.071,Y -433.665,Z 1892.496,A 0.000,B 0.000,C 90.000,E1 89.312} C_DIS
LIN {X -0.186,Y -425.340,Z 1892.489,A 0.000,B 0.000,C 90.000,E1 87.993} C_DIS
LIN {X -0.096,Y -411.877,Z 1892.477,A 0.000,B 0.000,C 90.000,E1 85.812} C_DIS
LIN {X -0.028,Y -401.710,Z 1892.467,A 0.000,B 0.000,C 90.000,E1 84.147} C_DIS
LIN {X -0.047,Y -389.746,Z 1892.457,A 0.000,B 0.000,C 90.000,E1 82.186} C_DIS
LIN {X 0.171,Y -377.840,Z 1892.445,A 0.000,B 0.000,C 90.000,E1 80.151} C_DIS
LIN {X 0.152,Y -361.201,Z 1892.429,A 0.000,B 0.000,C 90.000,E1 77.229} C_DIS
LIN {X -0.104,Y -345.597,Z 1892.412,A 0.000,B 0.000,C 90.000,E1 74.267} C_DIS
LIN {X -0.155,Y -333.632,Z 1892.399,A 0.000,B 0.000,C 90.000,E1 71.819} C_DIS
LIN {X 0.119,Y -321.935,Z 1892.385,A 0.000,B 0.000,C 90.000,E1 69.263} C_DIS
LIN {X -0.042,Y -309.309,Z 1892.369,A 0.000,B 0.000,C 90.000,E1 66.410} C_DIS
LIN {X 0.078,Y -299.791,Z 1892.356,A 0.000,B 0.000,C 90.000,E1 64.101} C_DIS
LIN {X -0.051,Y -287.731,Z 1892.340,A 0.000,B 0.000,C 90.000,E1 61.129} C_DIS
LIN {X -0.003,Y -278.301,Z 1892.326,A 0.000,B 0.000,C 90.000,E1 58.742} C_DIS
LIN {X 0.130,Y -268.816,Z 1892.313,A 0.000,B 0.000,C 90.000,E1 56.294} C_DIS
LIN {X 0.076,Y -260.601,Z 1892.301,A 0.000,B 0.000,C 90.000,E1 54.196} C_DIS
LIN {X 0.047,Y -250.997,Z 1892.287,A 0.000,B 0.000,C 90.000,E1 51.698} C_DIS
LIN {X -0.072,Y -241.440,Z 1892.273,A 0.000,B 0.000,C 90.000,E1 49.175} C_DIS
LIN {X -0.135,Y -230.794,Z 1892.257,A 0.000,B 0.000,C 90.000,E1 46.215} C_DIS
LIN {X 0.016,Y -220.581,Z 1892.240,A 0.000,B 0.000,C 90.000,E1 43.137} C_DIS
LIN {X 0.089,Y -210.953,Z 1892.222,A 0.000,B 0.000,C 90.000,E1 40.011} C_DIS
LIN {X -0.007,Y -202.163,Z 1892.205,A 0.000,B 0.000,C 90.000,E1 36.870} C_DIS
LIN {X -0.042,Y -194.185,Z 1892.187,A 0.000,B 0.000,C 90.000,E1 33.658} C_DIS
LIN {X -0.057,Y -186.948,Z 1892.169,A 0.000,B 0.000,C 90.000,E1 30.384} C_DIS
LIN {X -0.052,Y -180.421,Z 1892.150,A 0.000,B 0.000,C 90.000,E1 27.052} C_DIS
LIN {X -0.035,Y -175.995,Z 1892.136,A 0.000,B 0.000,C 90.000,E1 24.515} C_DIS
LIN {X -0.033,Y -170.836,Z 1892.117,A 0.000,B 0.000,C 90.000,E1 21.099} C_DIS
LIN {X -0.018,Y -166.457,Z 1892.098,A 0.000,B 0.000,C 90.000,E1 17.638} C_DIS
LIN {X 0.059,Y -162.880,Z 1892.079,A 0.000,B 0.000,C 90.000,E1 14.120} C_DIS
LIN {X 0.025,Y -159.262,Z 1892.054,A 0.000,B 0.000,C 90.000,E1 9.726} C_DIS
LIN {X -0.038,Y -156.425,Z 1892.024,A 0.000,B 0.000,C 90.000,E1 4.416} C_DIS
LIN {X -0.015,Y -154.186,Z 1891.982,A 0.000,B 0.000,C 90.000,E1 356.846} C_DIS
LIN {X 0.002,Y -155.140,Z 1891.923,A 0.000,B 0.000,C 90.000,E1 346.061} C_DIS
LIN {X 0.040,Y -157.428,Z 1891.893,A 0.000,B 0.000,C 90.000,E1 340.678} C_DIS
LIN {X 0.037,Y -160.565,Z 1891.868,A 0.000,B 0.000,C 90.000,E1 336.230} C_DIS
LIN {X 0.048,Y -164.000,Z 1891.848,A 0.000,B 0.000,C 90.000,E1 332.692} C_DIS
LIN {X 0.005,Y -168.434,Z 1891.829,A 0.000,B 0.000,C 90.000,E1 329.203} C_DIS
LIN {X 0.053,Y -173.843,Z 1891.810,A 0.000,B 0.000,C 90.000,E1 325.722} C_DIS
LIN {X -0.023,Y -178.596,Z 1891.795,A 0.000,B 0.000,C 90.000,E1 323.176} C_DIS
LIN {X -0.051,Y -184.162,Z 1891.781,A 0.000,B 0.000,C 90.000,E1 320.642} C_DIS
LIN {X 0.004,Y -190.629,Z 1891.767,A 0.000,B 0.000,C 90.000,E1 318.119} C_DIS
LIN {X 0.018,Y -198.105,Z 1891.754,A 0.000,B 0.000,C 90.000,E1 315.648} C_DIS
LIN {X 0.038,Y -206.530,Z 1891.740,A 0.000,B 0.000,C 90.000,E1 313.218} C_DIS
LIN {X -0.006,Y -217.484,Z 1891.725,A 0.000,B 0.000,C 90.000,E1 310.458} C_DIS
LIN {X 0.079,Y -229.457,Z 1891.710,A 0.000,B 0.000,C 90.000,E1 307.729} C_DIS
LIN {X -0.001,Y -244.286,Z 1891.693,A 0.000,B 0.000,C 90.000,E1 304.739} C_DIS
LIN {X -0.148,Y -258.053,Z 1891.679,A 0.000,B 0.000,C 90.000,E1 302.212} C_DIS
LIN {X 0.097,Y -272.110,Z 1891.665,A 0.000,B 0.000,C 90.000,E1 299.667} C_DIS
LIN {X 0.059,Y -280.238,Z 1891.657,A 0.000,B 0.000,C 90.000,E1 298.281} C_DIS
LIN {X -0.118,Y -292.974,Z 1891.646,A 0.000,B 0.000,C 90.000,E1 296.360} C_DIS
LIN {X -0.003,Y -306.217,Z 1891.635,A 0.000,B 0.000,C 90.000,E1 294.335} C_DIS
LIN {X 0.040,Y -317.038,Z 1891.626,A 0.000,B 0.000,C 90.000,E1 292.695} C_DIS
LIN {X 0.001,Y -327.482,Z 1891.617,A 0.000,B 0.000,C 90.000,E1 291.099} C_DIS
LIN {X 0.156,Y -335.347,Z 1891.610,A 0.000,B 0.000,C 90.000,E1 289.812} C_DIS
LIN {X -0.010,Y -340.961,Z 1891.605,A 0.000,B 0.000,C 90.000,E1 288.906} C_DIS
LIN {X -0.133,Y -346.213,Z 1891.600,A 0.000,B 0.000,C 90.000,E1 288.000} C_DIS
LIN {X 0.132,Y -350.941,Z 1891.595,A 0.000,B 0.000,C 90.000,E1 287.040} C_DIS
LIN {X 0.102,Y -354.996,Z 1891.590,A 0.000,B 0.000,C 90.000,E1 286.134} C_DIS
LIN {X 0.012,Y -358.536,Z 1891.585,A 0.000,B 0.000,C 90.000,E1 285.245} C_DIS
LIN {X -0.048,Y -361.438,Z 1891.580,A 0.000,B 0.000,C 90.000,E1 284.356} C_DIS
LIN {X -0.137,Y -363.060,Z 1891.576,A 0.000,B 0.000,C 90.000,E1 283.772} C_DIS
LIN {X -0.128,Y -364.314,Z 1891.573,A 0.000,B 0.000,C 90.000,E1 283.175} C_DIS
LIN {X 0.165,Y -365.114,Z 1891.570,A 0.000,B 0.000,C 90.000,E1 282.535} C_DIS
LIN {X 0.111,Y -365.616,Z 1891.567,A 0.000,B 0.000,C 90.000,E1 281.951} C_DIS
LIN {X 0.062,Y -365.648,Z 1891.563,A 0.000,B 0.000,C 90.000,E1 281.366} C_DIS
LIN {X 0.016,Y -365.363,Z 1891.560,A 0.000,B 0.000,C 90.000,E1 280.782} C_DIS
LIN {X -0.030,Y -364.675,Z 1891.557,A 0.000,B 0.000,C 90.000,E1 280.197} C_DIS
LIN {X -0.079,Y -363.620,Z 1891.553,A 0.000,B 0.000,C 90.000,E1 279.613} C_DIS
LIN {X -0.133,Y -362.187,Z 1891.550,A 0.000,B 0.000,C 90.000,E1 279.029} C_DIS
LIN {X 0.107,Y -360.448,Z 1891.547,A 0.000,B 0.000,C 90.000,E1 278.398} C_DIS
LIN {X -0.056,Y -357.204,Z 1891.542,A 0.000,B 0.000,C 90.000,E1 277.530} C_DIS
LIN {X -0.151,Y -354.606,Z 1891.538,A 0.000,B 0.000,C 90.000,E1 276.947} C_DIS
LIN {X -0.056,Y -349.874,Z 1891.533,A 0.000,B 0.000,C 90.000,E1 276.030} C_DIS
LIN {X 0.145,Y -346.117,Z 1891.530,A 0.000,B 0.000,C 90.000,E1 275.391} C_DIS
LIN {X -0.085,Y -341.732,Z 1891.527,A 0.000,B 0.000,C 90.000,E1 274.821} C_DIS
LIN {X 0.034,Y -336.723,Z 1891.523,A 0.000,B 0.000,C 90.000,E1 274.188} C_DIS
LIN {X 0.120,Y -330.985,Z 1891.520,A 0.000,B 0.000,C 90.000,E1 273.555} C_DIS
LIN {X 0.111,Y -324.871,Z 1891.517,A 0.000,B 0.000,C 90.000,E1 272.980} C_DIS
LIN {X 0.108,Y -318.624,Z 1891.514,A 0.000,B 0.000,C 90.000,E1 272.465} C_DIS
LIN {X 0.070,Y -312.196,Z 1891.511,A 0.000,B 0.000,C 90.000,E1 272.007} C_DIS
LIN {X 0.010,Y -305.371,Z 1891.509,A 0.000,B 0.000,C 90.000,E1 271.604} C_DIS
LIN {X -0.047,Y -297.999,Z 1891.507,A 0.000,B 0.000,C 90.000,E1 271.260} C_DIS
LIN {X -0.035,Y -290.512,Z 1891.505,A 0.000,B 0.000,C 90.000,E1 270.974} C_DIS
LIN {X 0.012,Y -282.670,Z 1891.504,A 0.000,B 0.000,C 90.000,E1 270.745} C_DIS
LIN {X 0.119,Y -267.709,Z 1891.502,A 0.000,B 0.000,C 90.000,E1 270.401} C_DIS
LIN {X -0.054,Y -256.257,Z 1891.501,A 0.000,B 0.000,C 90.000,E1 270.229} C_DIS
LIN {X -0.099,Y -247.440,Z 1891.500,A 0.000,B 0.000,C 90.000,E1 270.115} C_DIS
LIN {X 0.015,Y -236.769,Z 1891.500,A 0.000,B 0.000,C 90.000,E1 270.000} C_DIS
LIN {X -0.020,Y -181.560,Z 1891.500,A 0.000,B 0.000,C 90.000,E1 270.000} C_DIS
LIN {X 0.019,Y -180.836,Z 1891.472,A 0.000,B 0.000,C 90.000,E1 264.894} C_DIS
LIN {X -0.078,Y -178.943,Z 1891.443,A 0.000,B 0.000,C 90.000,E1 259.859} C_DIS
LIN {X -0.034,Y -175.994,Z 1891.415,A 0.000,B 0.000,C 90.000,E1 254.755} C_DIS
LIN {X -0.089,Y -175.498,Z 1891.411,A 0.000,B 0.000,C 90.000,E1 253.921} C_DIS
LIN {X -0.025,Y -172.240,Z 1891.387,A 0.000,B 0.000,C 90.000,E1 249.625} C_DIS
LIN {X -0.047,Y -171.718,Z 1891.382,A 0.000,B 0.000,C 90.000,E1 248.773} C_DIS
LIN {X -0.037,Y -167.313,Z 1891.353,A 0.000,B 0.000,C 90.000,E1 243.589} C_DIS
LIN {X 0.043,Y -166.694,Z 1891.348,A 0.000,B 0.000,C 90.000,E1 242.692} C_DIS
LIN {X 0.034,Y -162.676,Z 1891.324,A 0.000,B 0.000,C 90.000,E1 238.329} C_DIS
LIN {X 0.007,Y -161.366,Z 1891.314,A 0.000,B 0.000,C 90.000,E1 236.580} C_DIS
LIN {X -0.084,Y -157.360,Z 1891.290,A 0.000,B 0.000,C 90.000,E1 232.190} C_DIS
LIN {X 0.069,Y -155.349,Z 1891.275,A 0.000,B 0.000,C 90.000,E1 229.461} C_DIS
LIN {X -0.001,Y -151.694,Z 1891.250,A 0.000,B 0.000,C 90.000,E1 225.000} C_DIS
LIN {X 0.047,Y -150.556,Z 1891.240,A 0.000,B 0.000,C 90.000,E1 223.176} C_DIS
LIN {X -0.037,Y -147.283,Z 1891.215,A 0.000,B 0.000,C 90.000,E1 218.669} C_DIS
LIN {X -0.068,Y -145.311,Z 1891.194,A 0.000,B 0.000,C 90.000,E1 215.025} C_DIS
LIN {X 0.043,Y -142.401,Z 1891.164,A 0.000,B 0.000,C 90.000,E1 209.461} C_DIS
LIN {X 0.025,Y -141.383,Z 1891.148,A 0.000,B 0.000,C 90.000,E1 206.693} C_DIS
LIN {X 0.017,Y -139.350,Z 1891.112,A 0.000,B 0.000,C 90.000,E1 200.194} C_DIS
LIN {X 0.008,Y -138.788,Z 1891.097,A 0.000,B 0.000,C 90.000,E1 197.402} C_DIS
LIN {X 0.066,Y -138.345,Z 1891.055,A 0.000,B 0.000,C 90.000,E1 189.905} C_DIS
LIN {X -0.053,Y -139.385,Z 1891.008,A 0.000,B 0.000,C 90.000,E1 181.547} C_DIS
LIN {X 0.000,Y -141.281,Z 1890.972,A 0.000,B 0.000,C 90.000,E1 175.008} C_DIS
LIN {X -0.042,Y -142.645,Z 1890.957,A 0.000,B 0.000,C 90.000,E1 172.243} C_DIS
LIN {X 0.050,Y -144.980,Z 1890.931,A 0.000,B 0.000,C 90.000,E1 167.589} C_DIS
LIN {X 0.041,Y -147.607,Z 1890.911,A 0.000,B 0.000,C 90.000,E1 163.921} C_DIS
LIN {X -0.022,Y -150.229,Z 1890.891,A 0.000,B 0.000,C 90.000,E1 160.296} C_DIS
LIN {X -0.006,Y -153.620,Z 1890.870,A 0.000,B 0.000,C 90.000,E1 156.666} C_DIS
LIN {X -0.018,Y -157.035,Z 1890.850,A 0.000,B 0.000,C 90.000,E1 153.076} C_DIS
LIN {X -0.087,Y -161.160,Z 1890.831,A 0.000,B 0.000,C 90.000,E1 149.537} C_DIS
LIN {X -0.005,Y -163.256,Z 1890.821,A 0.000,B 0.000,C 90.000,E1 147.740} C_DIS
LIN {X 0.093,Y -167.694,Z 1890.801,A 0.000,B 0.000,C 90.000,E1 144.196} C_DIS
LIN {X 0.007,Y -171.515,Z 1890.787,A 0.000,B 0.000,C 90.000,E1 141.618} C_DIS
LIN {X 0.050,Y -176.452,Z 1890.768,A 0.000,B 0.000,C 90.000,E1 138.162} C_DIS
LIN {X -0.079,Y -180.748,Z 1890.753,A 0.000,B 0.000,C 90.000,E1 135.648} C_DIS
LIN {X 0.039,Y -186.153,Z 1890.735,A 0.000,B 0.000,C 90.000,E1 132.243} C_DIS
LIN {X -0.042,Y -190.791,Z 1890.721,A 0.000,B 0.000,C 90.000,E1 129.769} C_DIS
LIN {X 0.024,Y -196.547,Z 1890.703,A 0.000,B 0.000,C 90.000,E1 126.457} C_DIS
LIN {X -0.058,Y -201.319,Z 1890.689,A 0.000,B 0.000,C 90.000,E1 124.040} C_DIS
LIN {X 0.038,Y -207.291,Z 1890.671,A 0.000,B 0.000,C 90.000,E1 120.797} C_DIS
LIN {X 0.037,Y -210.546,Z 1890.662,A 0.000,B 0.000,C 90.000,E1 119.205} C_DIS
LIN {X 0.039,Y -216.350,Z 1890.645,A 0.000,B 0.000,C 90.000,E1 116.052} C_DIS
LIN {X -0.053,Y -219.487,Z 1890.636,A 0.000,B 0.000,C 90.000,E1 114.515} C_DIS
LIN {X -0.024,Y -224.123,Z 1890.621,A 0.000,B 0.000,C 90.000,E1 111.844} C_DIS
LIN {X -0.066,Y -283.391,Z 1890.621,A 0.000,B 0.000,C 90.000,E1 111.844} C_DIS
LIN {X 0.046,Y -286.148,Z 1890.621,A 0.000,B 0.000,C 90.000,E1 111.770} C_DIS
LIN {X 0.024,Y -289.759,Z 1890.620,A 0.000,B 0.000,C 90.000,E1 111.589} C_DIS
LIN {X 0.002,Y -291.961,Z 1890.619,A 0.000,B 0.000,C 90.000,E1 111.408} C_DIS
LIN {X -0.028,Y -295.837,Z 1890.616,A 0.000,B 0.000,C 90.000,E1 110.918} C_DIS
LIN {X 0.138,Y -311.095,Z 1890.601,A 0.000,B 0.000,C 90.000,E1 108.236} C_DIS
LIN {X -0.117,Y -325.845,Z 1890.589,A 0.000,B 0.000,C 90.000,E1 106.024} C_DIS
LIN {X -0.032,Y -339.686,Z 1890.578,A 0.000,B 0.000,C 90.000,E1 104.120} C_DIS
LIN {X -0.176,Y -354.715,Z 1890.568,A 0.000,B 0.000,C 90.000,E1 102.299} C_DIS
LIN {X -0.025,Y -373.192,Z 1890.557,A 0.000,B 0.000,C 90.000,E1 100.254} C_DIS
LIN {X 0.133,Y -392.064,Z 1890.547,A 0.000,B 0.000,C 90.000,E1 98.398} C_DIS
LIN {X 0.178,Y -411.347,Z 1890.537,A 0.000,B 0.000,C 90.000,E1 96.720} C_DIS
LIN {X 0.151,Y -433.760,Z 1890.528,A 0.000,B 0.000,C 90.000,E1 94.992} C_DIS
LIN {X 0.137,Y -439.392,Z 1890.526,A 0.000,B 0.000,C 90.000,E1 94.588} C_DIS
LIN {X 0.109,Y -443.354,Z 1890.523,A 0.000,B 0.000,C 90.000,E1 94.188} C_DIS
LIN {X -0.076,Y -445.048,Z 1890.522,A 0.000,B 0.000,C 90.000,E1 93.955} C_DIS
LIN {X 0.152,Y -446.338,Z 1890.521,A 0.000,B 0.000,C 90.000,E1 93.669} C_DIS
LIN {X 0.079,Y -448.027,Z 1890.518,A 0.000,B 0.000,C 90.000,E1 93.154} C_DIS
LIN {X 0.036,Y -448.680,Z 1890.515,A 0.000,B 0.000,C 90.000,E1 92.636} C_DIS
LIN {X -0.018,Y -448.401,Z 1890.512,A 0.000,B 0.000,C 90.000,E1 92.121} C_DIS
LIN {X -0.053,Y -447.156,Z 1890.509,A 0.000,B 0.000,C 90.000,E1 91.604} C_DIS
LIN {X 0.144,Y -446.113,Z 1890.507,A 0.000,B 0.000,C 90.000,E1 91.318} C_DIS
LIN {X -0.103,Y -444.725,Z 1890.506,A 0.000,B 0.000,C 90.000,E1 91.088} C_DIS
LIN {X -0.019,Y -431.562,Z 1890.494,A 0.000,B 0.000,C 90.000,E1 88.969} C_DIS
LIN {X -0.040,Y -421.496,Z 1890.485,A 0.000,B 0.000,C 90.000,E1 87.364} C_DIS
LIN {X -0.131,Y -409.717,Z 1890.475,A 0.000,B 0.000,C 90.000,E1 85.469} C_DIS
LIN {X -0.024,Y -397.826,Z 1890.464,A 0.000,B 0.000,C 90.000,E1 83.514} C_DIS
LIN {X -0.077,Y -385.856,Z 1890.453,A 0.000,B 0.000,C 90.000,E1 81.546} C_DIS
LIN {X 0.070,Y -373.994,Z 1890.442,A 0.000,B 0.000,C 90.000,E1 79.511} C_DIS
LIN {X -0.022,Y -355.965,Z 1890.424,A 0.000,B 0.000,C 90.000,E1 76.284} C_DIS
LIN {X -0.002,Y -342.157,Z 1890.409,A 0.000,B 0.000,C 90.000,E1 73.559} C_DIS
LIN {X -0.045,Y -330.278,Z 1890.395,A 0.000,B 0.000,C 90.000,E1 71.094} C_DIS
LIN {X 0.078,Y -317.243,Z 1890.379,A 0.000,B 0.000,C 90.000,E1 68.230} C_DIS
LIN {X -0.094,Y -304.842,Z 1890.363,A 0.000,B 0.000,C 90.000,E1 65.357} C_DIS
LIN {X -0.082,Y -295.315,Z 1890.350,A 0.000,B 0.000,C 90.000,E1 63.050} C_DIS
LIN {X 0.116,Y -286.002,Z 1890.337,A 0.000,B 0.000,C 90.000,E1 60.667} C_DIS
LIN {X -0.115,Y -276.567,Z 1890.324,A 0.000,B 0.000,C 90.000,E1 58.329} C_DIS
LIN {X -0.015,Y -267.084,Z 1890.310,A 0.000,B 0.000,C 90.000,E1 55.881} C_DIS
LIN {X -0.051,Y -257.466,Z 1890.297,A 0.000,B 0.000,C 90.000,E1 53.417} C_DIS
LIN {X 0.012,Y -247.868,Z 1890.283,A 0.000,B 0.000,C 90.000,E1 50.884} C_DIS
LIN {X -0.036,Y -237.026,Z 1890.266,A 0.000,B 0.000,C 90.000,E1 47.957} C_DIS
LIN {X -0.114,Y -225.290,Z 1890.248,A 0.000,B 0.000,C 90.000,E1 44.595} C_DIS
LIN {X 0.127,Y -214.146,Z 1890.228,A 0.000,B 0.000,C 90.000,E1 41.067} C_DIS
LIN {X 0.065,Y -205.023,Z 1890.211,A 0.000,B 0.000,C 90.000,E1 37.935} C_DIS
LIN {X 0.038,Y -196.805,Z 1890.193,A 0.000,B 0.000,C 90.000,E1 34.739} C_DIS
LIN {X 0.083,Y -189.316,Z 1890.175,A 0.000,B 0.000,C 90.000,E1 31.465} C_DIS
LIN {X 0.071,Y -182.559,Z 1890.156,A 0.000,B 0.000,C 90.000,E1 28.153} C_DIS
LIN {X -0.039,Y -176.496,Z 1890.138,A 0.000,B 0.000,C 90.000,E1 24.823} C_DIS
LIN {X -0.026,Y -171.269,Z 1890.119,A 0.000,B 0.000,C 90.000,E1 21.408} C_DIS
LIN {X 0.000,Y -166.811,Z 1890.100,A 0.000,B 0.000,C 90.000,E1 17.946} C_DIS
LIN {X -0.067,Y -163.170,Z 1890.080,A 0.000,B 0.000,C 90.000,E1 14.481} C_DIS
LIN {X -0.053,Y -159.470,Z 1890.056,A 0.000,B 0.000,C 90.000,E1 10.074} C_DIS
LIN {X -0.024,Y -156.953,Z 1890.031,A 0.000,B 0.000,C 90.000,E1 5.625} C_DIS
LIN {X -0.028,Y -154.708,Z 1889.997,A 0.000,B 0.000,C 90.000,E1 359.542} C_DIS
LIN {X 0.051,Y -154.204,Z 1889.943,A 0.000,B 0.000,C 90.000,E1 349.634} C_DIS
LIN {X -0.013,Y -156.102,Z 1889.908,A 0.000,B 0.000,C 90.000,E1 343.378} C_DIS
LIN {X 0.021,Y -158.524,Z 1889.883,A 0.000,B 0.000,C 90.000,E1 338.901} C_DIS
LIN {X 0.033,Y -162.143,Z 1889.858,A 0.000,B 0.000,C 90.000,E1 334.460} C_DIS
LIN {X 0.085,Y -166.107,Z 1889.839,A 0.000,B 0.000,C 90.000,E1 330.923} C_DIS
LIN {X 0.017,Y -169.704,Z 1889.824,A 0.000,B 0.000,C 90.000,E1 328.329} C_DIS
LIN {X 0.051,Y -173.850,Z 1889.810,A 0.000,B 0.000,C 90.000,E1 325.722} C_DIS
LIN {X -0.024,Y -178.604,Z 1889.795,A 0.000,B 0.000,C 90.000,E1 323.176} C_DIS
LIN {X -0.051,Y -184.171,Z 1889.781,A 0.000,B 0.000,C 90.000,E1 320.642} C_DIS
LIN {X 0.004,Y -190.638,Z 1889.767,A 0.000,B 0.000,C 90.000,E1 318.119} C_DIS
LIN {X 0.018,Y -198.111,Z 1889.754,A 0.000,B 0.000,C 90.000,E1 315.648} C_DIS
LIN {X 0.038,Y -206.536,Z 1889.740,A 0.000,B 0.000,C 90.000,E1 313.218} C_DIS
LIN {X -0.006,Y -217.492,Z 1889.725,A 0.000,B 0.000,C 90.000,E1 310.458} C_DIS
LIN {X 0.079,Y -229.466,Z 1889.710,A 0.000,B 0.000,C 90.000,E1 307.729} C_DIS
LIN {X 0.000,Y -244.296,Z 1889.693,A 0.000,B 0.000,C 90.000,E1 304.739} C_DIS
LIN {X -0.148,Y -258.063,Z 1889.679,A 0.000,B 0.000,C 90.000,E1 302.212} C_DIS
LIN {X 0.097,Y -272.119,Z 1889.665,A 0.000,B 0.000,C 90.000,E1 299.667} C_DIS
LIN {X -0.047,Y -280.267,Z 1889.657,A 0.000,B 0.000,C 90.000,E1 298.359} C_DIS
LIN {X 0.113,Y -291.434,Z 1889.648,A 0.000,B 0.000,C 90.000,E1 296.616} C_DIS
LIN {X -0.068,Y -304.731,Z 1889.637,A 0.000,B 0.000,C 90.000,E1 294.643} C_DIS
LIN {X -0.059,Y -315.674,Z 1889.628,A 0.000,B 0.000,C 90.000,E1 293.003} C_DIS
LIN {X -0.117,Y -326.187,Z 1889.619,A 0.000,B 0.000,C 90.000,E1 291.408} C_DIS
LIN {X 0.018,Y -334.254,Z 1889.612,A 0.000,B 0.000,C 90.000,E1 290.120} C_DIS
LIN {X -0.175,Y -341.784,Z 1889.605,A 0.000,B 0.000,C 90.000,E1 288.906} C_DIS
LIN {X 0.038,Y -347.030,Z 1889.600,A 0.000,B 0.000,C 90.000,E1 287.946} C_DIS
LIN {X -0.021,Y -351.733,Z 1889.595,A 0.000,B 0.000,C 90.000,E1 287.040} C_DIS
LIN {X -0.046,Y -355.752,Z 1889.590,A 0.000,B 0.000,C 90.000,E1 286.134} C_DIS
LIN {X -0.131,Y -359.272,Z 1889.585,A 0.000,B 0.000,C 90.000,E1 285.245} C_DIS
LIN {X 0.166,Y -362.131,Z 1889.580,A 0.000,B 0.000,C 90.000,E1 284.300} C_DIS
LIN {X 0.084,Y -363.744,Z 1889.576,A 0.000,B 0.000,C 90.000,E1 283.716} C_DIS
LIN {X 0.100,Y -364.887,Z 1889.573,A 0.000,B 0.000,C 90.000,E1 283.119} C_DIS
LIN {X 0.040,Y -365.720,Z 1889.570,A 0.000,B 0.000,C 90.000,E1 282.535} C_DIS
LIN {X -0.011,Y -366.140,Z 1889.566,A 0.000,B 0.000,C 90.000,E1 281.951} C_DIS
LIN {X -0.056,Y -366.174,Z 1889.563,A 0.000,B 0.000,C 90.000,E1 281.366} C_DIS
LIN {X -0.098,Y -365.837,Z 1889.560,A 0.000,B 0.000,C 90.000,E1 280.782} C_DIS
LIN {X -0.141,Y -365.102,Z 1889.557,A 0.000,B 0.000,C 90.000,E1 280.197} C_DIS
LIN {X 0.173,Y -363.999,Z 1889.553,A 0.000,B 0.000,C 90.000,E1 279.557} C_DIS
LIN {X 0.119,Y -362.536,Z 1889.550,A 0.000,B 0.000,C 90.000,E1 278.973} C_DIS
LIN {X 0.005,Y -360.762,Z 1889.547,A 0.000,B 0.000,C 90.000,E1 278.398} C_DIS
LIN {X -0.154,Y -357.485,Z 1889.542,A 0.000,B 0.000,C 90.000,E1 277.530} C_DIS
LIN {X 0.106,Y -354.860,Z 1889.538,A 0.000,B 0.000,C 90.000,E1 276.891} C_DIS
LIN {X -0.111,Y -350.045,Z 1889.533,A 0.000,B 0.000,C 90.000,E1 276.024} C_DIS
LIN {X 0.056,Y -346.259,Z 1889.530,A 0.000,B 0.000,C 90.000,E1 275.391} C_DIS
LIN {X -0.143,Y -341.846,Z 1889.527,A 0.000,B 0.000,C 90.000,E1 274.816} C_DIS
LIN {X -0.051,Y -336.762,Z 1889.523,A 0.000,B 0.000,C 90.000,E1 274.188} C_DIS
LIN {X 0.044,Y -331.010,Z 1889.520,A 0.000,B 0.000,C 90.000,E1 273.555} C_DIS
LIN {X 0.077,Y -324.982,Z 1889.517,A 0.000,B 0.000,C 90.000,E1 272.980} C_DIS
LIN {X 0.035,Y -318.612,Z 1889.514,A 0.000,B 0.000,C 90.000,E1 272.465} C_DIS
LIN {X -0.002,Y -312.068,Z 1889.511,A 0.000,B 0.000,C 90.000,E1 272.007} C_DIS
LIN {X -0.026,Y -305.380,Z 1889.509,A 0.000,B 0.000,C 90.000,E1 271.604} C_DIS
LIN {X -0.078,Y -298.078,Z 1889.507,A 0.000,B 0.000,C 90.000,E1 271.260} C_DIS
LIN {X -0.092,Y -290.194,Z 1889.505,A 0.000,B 0.000,C 90.000,E1 270.974} C_DIS
LIN {X -0.027,Y -282.242,Z 1889.504,A 0.000,B 0.000,C 90.000,E1 270.745} C_DIS
LIN {X 0.063,Y -263.964,Z 1889.502,A 0.000,B 0.000,C 90.000,E1 270.344} C_DIS
LIN {X 0.088,Y -249.140,Z 1889.500,A 0.000,B 0.000,C 90.000,E1 270.057} C_DIS
LIN {X -0.102,Y -236.805,Z 1889.500,A 0.000,B 0.000,C 90.000,E1 269.943} C_DIS
LIN {X 0.065,Y -232.348,Z 1889.500,A 0.000,B 0.000,C 90.000,E1 269.885} C_DIS
LIN {X 0.024,Y -181.540,Z 1889.499,A 0.000,B 0.000,C 90.000,E1 269.885} C_DIS
LIN {X -0.041,Y -180.905,Z 1889.474,A 0.000,B 0.000,C 90.000,E1 265.355} C_DIS
LIN {X 0.033,Y -180.675,Z 1889.469,A 0.000,B 0.000,C 90.000,E1 264.489} C_DIS
LIN {X -0.068,Y -178.757,Z 1889.441,A 0.000,B 0.000,C 90.000,E1 259.454} C_DIS
LIN {X 0.004,Y -175.804,Z 1889.413,A 0.000,B 0.000,C 90.000,E1 254.338} C_DIS
LIN {X -0.001,Y -171.990,Z 1889.385,A 0.000,B 0.000,C 90.000,E1 249.209} C_DIS
LIN {X 0.037,Y -171.399,Z 1889.380,A 0.000,B 0.000,C 90.000,E1 248.337} C_DIS
LIN {X 0.021,Y -167.641,Z 1889.356,A 0.000,B 0.000,C 90.000,E1 244.024} C_DIS
LIN {X 0.037,Y -166.301,Z 1889.346,A 0.000,B 0.000,C 90.000,E1 242.281} C_DIS
LIN {X 0.030,Y -163.047,Z 1889.327,A 0.000,B 0.000,C 90.000,E1 238.791} C_DIS
LIN {X -0.008,Y -160.979,Z 1889.312,A 0.000,B 0.000,C 90.000,E1 236.167} C_DIS
LIN {X -0.031,Y -157.729,Z 1889.292,A 0.000,B 0.000,C 90.000,E1 232.637} C_DIS
LIN {X -0.092,Y -155.768,Z 1889.278,A 0.000,B 0.000,C 90.000,E1 229.989} C_DIS
LIN {X -0.036,Y -152.023,Z 1889.253,A 0.000,B 0.000,C 90.000,E1 225.486} C_DIS
LIN {X -0.019,Y -150.271,Z 1889.238,A 0.000,B 0.000,C 90.000,E1 222.771} C_DIS
LIN {X -0.001,Y -147.023,Z 1889.212,A 0.000,B 0.000,C 90.000,E1 218.222} C_DIS
LIN {X 0.021,Y -145.605,Z 1889.197,A 0.000,B 0.000,C 90.000,E1 215.471} C_DIS
LIN {X 0.024,Y -142.991,Z 1889.172,A 0.000,B 0.000,C 90.000,E1 210.875} C_DIS
LIN {X 0.024,Y -141.618,Z 1889.151,A 0.000,B 0.000,C 90.000,E1 207.180} C_DIS
LIN {X 0.065,Y -139.430,Z 1889.115,A 0.000,B 0.000,C 90.000,E1 200.663} C_DIS
LIN {X -0.061,Y -139.160,Z 1889.105,A 0.000,B 0.000,C 90.000,E1 198.852} C_DIS
LIN {X -0.023,Y -138.342,Z 1889.058,A 0.000,B 0.000,C 90.000,E1 190.433} C_DIS
LIN {X -0.016,Y -139.480,Z 1889.006,A 0.000,B 0.000,C 90.000,E1 181.088} C_DIS
LIN {X 0.065,Y -141.068,Z 1888.975,A 0.000,B 0.000,C 90.000,E1 175.469} C_DIS
LIN {X 0.019,Y -142.443,Z 1888.959,A 0.000,B 0.000,C 90.000,E1 172.704} C_DIS
LIN {X -0.032,Y -144.682,Z 1888.934,A 0.000,B 0.000,C 90.000,E1 168.105} C_DIS
LIN {X 0.063,Y -147.272,Z 1888.913,A 0.000,B 0.000,C 90.000,E1 164.393} C_DIS
LIN {X -0.062,Y -150.590,Z 1888.888,A 0.000,B 0.000,C 90.000,E1 159.880} C_DIS
LIN {X 0.016,Y -154.062,Z 1888.868,A 0.000,B 0.000,C 90.000,E1 156.230} C_DIS
LIN {X 0.082,Y -157.481,Z 1888.848,A 0.000,B 0.000,C 90.000,E1 152.615} C_DIS
LIN {X 0.028,Y -161.706,Z 1888.828,A 0.000,B 0.000,C 90.000,E1 149.076} C_DIS
LIN {X 0.042,Y -165.900,Z 1888.809,A 0.000,B 0.000,C 90.000,E1 145.548} C_DIS
LIN {X 0.029,Y -170.884,Z 1888.789,A 0.000,B 0.000,C 90.000,E1 142.065} C_DIS
LIN {X 0.057,Y -175.752,Z 1888.770,A 0.000,B 0.000,C 90.000,E1 138.609} C_DIS
LIN {X -0.070,Y -181.362,Z 1888.751,A 0.000,B 0.000,C 90.000,E1 135.243} C_DIS
LIN {X 0.064,Y -186.855,Z 1888.733,A 0.000,B 0.000,C 90.000,E1 131.838} C_DIS
LIN {X 0.017,Y -191.439,Z 1888.719,A 0.000,B 0.000,C 90.000,E1 129.358} C_DIS
LIN {X -0.050,Y -197.292,Z 1888.700,A 0.000,B 0.000,C 90.000,E1 126.091} C_DIS
LIN {X -0.014,Y -200.570,Z 1888.691,A 0.000,B 0.000,C 90.000,E1 124.452} C_DIS
LIN {X 0.063,Y -206.453,Z 1888.673,A 0.000,B 0.000,C 90.000,E1 121.209} C_DIS
LIN {X 0.055,Y -209.738,Z 1888.665,A 0.000,B 0.000,C 90.000,E1 119.617} C_DIS
LIN {X -0.108,Y -217.101,Z 1888.643,A 0.000,B 0.000,C 90.000,E1 115.720} C_DIS
LIN {X 0.042,Y -218.727,Z 1888.638,A 0.000,B 0.000,C 90.000,E1 114.899} C_DIS
LIN {X -0.026,Y -224.123,Z 1888.621,A 0.000,B 0.000,C 90.000,E1 111.844} C_DIS
LIN {X -0.065,Y -283.570,Z 1888.621,A 0.000,B 0.000,C 90.000,E1 111.844} C_DIS
LIN {X -0.159,Y -284.945,Z 1888.621,A 0.000,B 0.000,C 90.000,E1 111.844} C_DIS
LIN {X -0.143,Y -288.263,Z 1888.620,A 0.000,B 0.000,C 90.000,E1 111.716} C_DIS
LIN {X -0.042,Y -291.494,Z 1888.619,A 0.000,B 0.000,C 90.000,E1 111.461} C_DIS
LIN {X -0.153,Y -295.173,Z 1888.617,A 0.000,B 0.000,C 90.000,E1 111.046} C_DIS
LIN {X 0.042,Y -306.403,Z 1888.606,A 0.000,B 0.000,C 90.000,E1 109.033} C_DIS
LIN {X 0.178,Y -320.670,Z 1888.593,A 0.000,B 0.000,C 90.000,E1 106.732} C_DIS
LIN {X 0.172,Y -334.061,Z 1888.583,A 0.000,B 0.000,C 90.000,E1 104.828} C_DIS
LIN {X -0.077,Y -348.614,Z 1888.572,A 0.000,B 0.000,C 90.000,E1 103.008} C_DIS
LIN {X 0.090,Y -364.214,Z 1888.562,A 0.000,B 0.000,C 90.000,E1 101.186} C_DIS
LIN {X 0.090,Y -382.924,Z 1888.552,A 0.000,B 0.000,C 90.000,E1 99.265} C_DIS
LIN {X 0.016,Y -401.996,Z 1888.542,A 0.000,B 0.000,C 90.000,E1 97.530} C_DIS
LIN {X -0.121,Y -424.237,Z 1888.532,A 0.000,B 0.000,C 90.000,E1 95.739} C_DIS
LIN {X -0.160,Y -438.356,Z 1888.526,A 0.000,B 0.000,C 90.000,E1 94.702} C_DIS
LIN {X -0.149,Y -442.705,Z 1888.524,A 0.000,B 0.000,C 90.000,E1 94.302} C_DIS
LIN {X 0.155,Y -445.795,Z 1888.521,A 0.000,B 0.000,C 90.000,E1 93.784} C_DIS
LIN {X 0.066,Y -447.745,Z 1888.518,A 0.000,B 0.000,C 90.000,E1 93.269} C_DIS
LIN {X 0.020,Y -448.606,Z 1888.515,A 0.000,B 0.000,C 90.000,E1 92.751} C_DIS
LIN {X -0.036,Y -448.524,Z 1888.512,A 0.000,B 0.000,C 90.000,E1 92.236} C_DIS
LIN {X -0.071,Y -447.496,Z 1888.510,A 0.000,B 0.000,C 90.000,E1 91.718} C_DIS
LIN {X -0.121,Y -445.353,Z 1888.507,A 0.000,B 0.000,C 90.000,E1 91.203} C_DIS
LIN {X -0.176,Y -433.896,Z 1888.496,A 0.000,B 0.000,C 90.000,E1 89.370} C_DIS
LIN {X -0.152,Y -423.898,Z 1888.487,A 0.000,B 0.000,C 90.000,E1 87.764} C_DIS
LIN {X -0.181,Y -412.119,Z 1888.477,A 0.000,B 0.000,C 90.000,E1 85.869} C_DIS
LIN {X -0.105,Y -401.956,Z 1888.468,A 0.000,B 0.000,C 90.000,E1 84.204} C_DIS
LIN {X -0.121,Y -389.987,Z 1888.457,A 0.000,B 0.000,C 90.000,E1 82.243} C_DIS
LIN {X 0.112,Y -378.082,Z 1888.446,A 0.000,B 0.000,C 90.000,E1 80.208} C_DIS
LIN {X 0.025,Y -361.426,Z 1888.429,A 0.000,B 0.000,C 90.000,E1 77.297} C_DIS
LIN {X 0.102,Y -345.808,Z 1888.413,A 0.000,B 0.000,C 90.000,E1 74.283} C_DIS
LIN {X 0.139,Y -333.832,Z 1888.399,A 0.000,B 0.000,C 90.000,E1 71.819} C_DIS
LIN {X -0.008,Y -322.129,Z 1888.385,A 0.000,B 0.000,C 90.000,E1 69.337} C_DIS
LIN {X -0.171,Y -309.483,Z 1888.369,A 0.000,B 0.000,C 90.000,E1 66.485} C_DIS
LIN {X 0.086,Y -299.967,Z 1888.356,A 0.000,B 0.000,C 90.000,E1 64.152} C_DIS
LIN {X -0.037,Y -287.892,Z 1888.340,A 0.000,B 0.000,C 90.000,E1 61.179} C_DIS
LIN {X 0.025,Y -278.476,Z 1888.327,A 0.000,B 0.000,C 90.000,E1 58.791} C_DIS
LIN {X 0.013,Y -268.987,Z 1888.313,A 0.000,B 0.000,C 90.000,E1 56.373} C_DIS
LIN {X -0.037,Y -260.782,Z 1888.302,A 0.000,B 0.000,C 90.000,E1 54.276} C_DIS
LIN {X 0.100,Y -251.180,Z 1888.288,A 0.000,B 0.000,C 90.000,E1 51.743} C_DIS
LIN {X -0.014,Y -241.618,Z 1888.273,A 0.000,B 0.000,C 90.000,E1 49.218} C_DIS
LIN {X 0.100,Y -230.961,Z 1888.257,A 0.000,B 0.000,C 90.000,E1 46.215} C_DIS
LIN {X -0.068,Y -220.740,Z 1888.240,A 0.000,B 0.000,C 90.000,E1 43.218} C_DIS
LIN {X 0.013,Y -211.101,Z 1888.223,A 0.000,B 0.000,C 90.000,E1 40.092} C_DIS
LIN {X 0.035,Y -203.336,Z 1888.207,A 0.000,B 0.000,C 90.000,E1 37.317} C_DIS
LIN {X -0.020,Y -195.264,Z 1888.190,A 0.000,B 0.000,C 90.000,E1 34.119} C_DIS
LIN {X -0.012,Y -187.922,Z 1888.171,A 0.000,B 0.000,C 90.000,E1 30.846} C_DIS
LIN {X 0.015,Y -181.301,Z 1888.153,A 0.000,B 0.000,C 90.000,E1 27.513} C_DIS
LIN {X 0.037,Y -175.396,Z 1888.134,A 0.000,B 0.000,C 90.000,E1 24.131} C_DIS
LIN {X -0.042,Y -170.323,Z 1888.115,A 0.000,B 0.000,C 90.000,E1 20.737} C_DIS
LIN {X -0.038,Y -166.036,Z 1888.096,A 0.000,B 0.000,C 90.000,E1 17.275} C_DIS
LIN {X -0.013,Y -162.527,Z 1888.077,A 0.000,B 0.000,C 90.000,E1 13.772} C_DIS
LIN {X -0.028,Y -159.597,Z 1888.057,A 0.000,B 0.000,C 90.000,E1 10.254} C_DIS
LIN {X 0.027,Y -157.030,Z 1888.032,A 0.000,B 0.000,C 90.000,E1 5.796} C_DIS
LIN {X 0.000,Y -154.835,Z 1888.000,A 0.000,B 0.000,C 90.000,E1 360.000} C_DIS
LIN {X -0.015,Y -154.080,Z 1887.948,A 0.000,B 0.000,C 90.000,E1 350.557} C_DIS
LIN {X -0.013,Y -156.098,Z 1887.908,A 0.000,B 0.000,C 90.000,E1 343.378} C_DIS
LIN {X 0.020,Y -158.521,Z 1887.883,A 0.000,B 0.000,C 90.000,E1 338.901} C_DIS
LIN {X 0.032,Y -162.144,Z 1887.858,A 0.000,B 0.000,C 90.000,E1 334.460} C_DIS
LIN {X 0.084,Y -166.109,Z 1887.839,A 0.000,B 0.000,C 90.000,E1 330.923} C_DIS
LIN {X 0.016,Y -169.709,Z 1887.824,A 0.000,B 0.000,C 90.000,E1 328.329} C_DIS
LIN {X 0.051,Y -173.856,Z 1887.810,A 0.000,B 0.000,C 90.000,E1 325.722} C_DIS
LIN {X -0.025,Y -178.611,Z 1887.795,A 0.000,B 0.000,C 90.000,E1 323.176} C_DIS
LIN {X -0.051,Y -184.178,Z 1887.781,A 0.000,B 0.000,C 90.000,E1 320.642} C_DIS
LIN {X -0.065,Y -187.734,Z 1887.773,A 0.000,B 0.000,C 90.000,E1 319.218} C_DIS
LIN {X 0.056,Y -189.137,Z 1887.773,A 0.000,B 0.000,C 90.000,E1 319.175} C_DIS
LIN {X -0.052,Y -189.838,Z 1887.773,A 0.000,B 0.000,C 90.000,E1 319.175} C_DIS
LIN {X 0.061,Y -191.546,Z 1887.772,A 0.000,B 0.000,C 90.000,E1 318.933} C_DIS
LIN {X -0.056,Y -194.676,Z 1887.768,A 0.000,B 0.000,C 90.000,E1 318.243} C_DIS
LIN {X 0.044,Y -197.316,Z 1887.763,A 0.000,B 0.000,C 90.000,E1 317.391} C_DIS
LIN {X -0.111,Y -201.854,Z 1887.754,A 0.000,B 0.000,C 90.000,E1 315.810} C_DIS
LIN {X -0.117,Y -210.753,Z 1887.737,A 0.000,B 0.000,C 90.000,E1 312.609} C_DIS
LIN {X 0.050,Y -215.792,Z 1887.728,A 0.000,B 0.000,C 90.000,E1 310.987} C_DIS
LIN {X 0.086,Y -220.169,Z 1887.721,A 0.000,B 0.000,C 90.000,E1 309.806} C_DIS
LIN {X -0.066,Y -232.968,Z 1887.706,A 0.000,B 0.000,C 90.000,E1 307.030} C_DIS
LIN {X -0.060,Y -248.040,Z 1887.689,A 0.000,B 0.000,C 90.000,E1 304.040} C_DIS
LIN {X -0.155,Y -259.931,Z 1887.677,A 0.000,B 0.000,C 90.000,E1 301.878} C_DIS
LIN {X -0.022,Y -272.143,Z 1887.665,A 0.000,B 0.000,C 90.000,E1 299.716} C_DIS
LIN {X 0.153,Y -287.624,Z 1887.652,A 0.000,B 0.000,C 90.000,E1 297.257} C_DIS
LIN {X -0.097,Y -300.950,Z 1887.640,A 0.000,B 0.000,C 90.000,E1 295.283} C_DIS
LIN {X -0.137,Y -312.007,Z 1887.631,A 0.000,B 0.000,C 90.000,E1 293.643} C_DIS
LIN {X -0.064,Y -320.613,Z 1887.624,A 0.000,B 0.000,C 90.000,E1 292.333} C_DIS
LIN {X 0.001,Y -328.996,Z 1887.617,A 0.000,B 0.000,C 90.000,E1 291.046} C_DIS
LIN {X -0.138,Y -336.956,Z 1887.610,A 0.000,B 0.000,C 90.000,E1 289.812} C_DIS
LIN {X 0.023,Y -342.574,Z 1887.605,A 0.000,B 0.000,C 90.000,E1 288.852} C_DIS
LIN {X -0.077,Y -347.811,Z 1887.600,A 0.000,B 0.000,C 90.000,E1 287.946} C_DIS
LIN {X -0.136,Y -352.462,Z 1887.594,A 0.000,B 0.000,C 90.000,E1 287.040} C_DIS
LIN {X 0.192,Y -356.492,Z 1887.589,A 0.000,B 0.000,C 90.000,E1 286.079} C_DIS
LIN {X 0.114,Y -359.966,Z 1887.584,A 0.000,B 0.000,C 90.000,E1 285.190} C_DIS
LIN {X 0.113,Y -361.964,Z 1887.581,A 0.000,B 0.000,C 90.000,E1 284.592} C_DIS
LIN {X 0.027,Y -363.647,Z 1887.578,A 0.000,B 0.000,C 90.000,E1 284.008} C_DIS
LIN {X 0.041,Y -365.003,Z 1887.575,A 0.000,B 0.000,C 90.000,E1 283.411} C_DIS
LIN {X -0.020,Y -365.977,Z 1887.571,A 0.000,B 0.000,C 90.000,E1 282.827} C_DIS
LIN {X -0.072,Y -366.545,Z 1887.568,A 0.000,B 0.000,C 90.000,E1 282.243} C_DIS
LIN {X -0.115,Y -366.727,Z 1887.565,A 0.000,B 0.000,C 90.000,E1 281.658} C_DIS
LIN {X -0.155,Y -366.555,Z 1887.561,A 0.000,B 0.000,C 90.000,E1 281.074} C_DIS
LIN {X -0.194,Y -365.969,Z 1887.558,A 0.000,B 0.000,C 90.000,E1 280.489} C_DIS
LIN {X 0.125,Y -365.006,Z 1887.555,A 0.000,B 0.000,C 90.000,E1 279.849} C_DIS
LIN {X 0.079,Y -363.686,Z 1887.552,A 0.000,B 0.000,C 90.000,E1 279.265} C_DIS
LIN {X 0.025,Y -362.005,Z 1887.548,A 0.000,B 0.000,C 90.000,E1 278.681} C_DIS
LIN {X -0.128,Y -358.972,Z 1887.543,A 0.000,B 0.000,C 90.000,E1 277.814} C_DIS
LIN {X 0.047,Y -355.119,Z 1887.538,A 0.000,B 0.000,C 90.000,E1 276.891} C_DIS
LIN {X -0.106,Y -352.018,Z 1887.535,A 0.000,B 0.000,C 90.000,E1 276.315} C_DIS
LIN {X 0.074,Y -348.442,Z 1887.532,A 0.000,B 0.000,C 90.000,E1 275.682} C_DIS
LIN {X -0.113,Y -344.306,Z 1887.528,A 0.000,B 0.000,C 90.000,E1 275.106} C_DIS
LIN {X 0.021,Y -339.537,Z 1887.525,A 0.000,B 0.000,C 90.000,E1 274.473} C_DIS
LIN {X 0.123,Y -334.050,Z 1887.521,A 0.000,B 0.000,C 90.000,E1 273.841} C_DIS
LIN {X 0.029,Y -328.185,Z 1887.518,A 0.000,B 0.000,C 90.000,E1 273.269} C_DIS
LIN {X -0.108,Y -322.017,Z 1887.515,A 0.000,B 0.000,C 90.000,E1 272.751} C_DIS
LIN {X 0.057,Y -315.734,Z 1887.512,A 0.000,B 0.000,C 90.000,E1 272.236} C_DIS
LIN {X 0.143,Y -308.989,Z 1887.510,A 0.000,B 0.000,C 90.000,E1 271.776} C_DIS
LIN {X -0.069,Y -301.945,Z 1887.508,A 0.000,B 0.000,C 90.000,E1 271.432} C_DIS
LIN {X 0.078,Y -294.536,Z 1887.506,A 0.000,B 0.000,C 90.000,E1 271.088} C_DIS
LIN {X -0.003,Y -286.833,Z 1887.505,A 0.000,B 0.000,C 90.000,E1 270.859} C_DIS
LIN {X 0.095,Y -275.527,Z 1887.503,A 0.000,B 0.000,C 90.000,E1 270.573} C_DIS
LIN {X -0.066,Y -250.367,Z 1887.501,A 0.000,B 0.000,C 90.000,E1 270.115} C_DIS
LIN {X 0.056,Y -238.323,Z 1887.499,A 0.000,B 0.000,C 90.000,E1 269.885} C_DIS
LIN {X 0.029,Y -230.690,Z 1887.499,A 0.000,B 0.000,C 90.000,E1 269.828} C_DIS
LIN {X -0.009,Y -227.452,Z 1887.499,A 0.000,B 0.000,C 90.000,E1 269.828} C_DIS
LIN {X -0.036,Y -181.523,Z 1887.499,A 0.000,B 0.000,C 90.000,E1 269.828} C_DIS
LIN {X 0.073,Y -180.907,Z 1887.475,A 0.000,B 0.000,C 90.000,E1 265.527} C_DIS
LIN {X -0.049,Y -180.771,Z 1887.471,A 0.000,B 0.000,C 90.000,E1 264.723} C_DIS
LIN {X 0.022,Y -178.866,Z 1887.443,A 0.000,B 0.000,C 90.000,E1 259.634} C_DIS
LIN {X -0.077,Y -175.909,Z 1887.414,A 0.000,B 0.000,C 90.000,E1 254.574} C_DIS
LIN {X -0.020,Y -174.594,Z 1887.405,A 0.000,B 0.000,C 90.000,E1 252.851} C_DIS
LIN {X 0.066,Y -171.576,Z 1887.381,A 0.000,B 0.000,C 90.000,E1 248.539} C_DIS
LIN {X 0.047,Y -167.799,Z 1887.357,A 0.000,B 0.000,C 90.000,E1 244.229} C_DIS
LIN {X 0.062,Y -166.518,Z 1887.347,A 0.000,B 0.000,C 90.000,E1 242.487} C_DIS
LIN {X 0.050,Y -162.518,Z 1887.323,A 0.000,B 0.000,C 90.000,E1 238.122} C_DIS
LIN {X 0.021,Y -161.191,Z 1887.313,A 0.000,B 0.000,C 90.000,E1 236.373} C_DIS
LIN {X -0.076,Y -157.202,Z 1887.289,A 0.000,B 0.000,C 90.000,E1 231.984} C_DIS
LIN {X -0.053,Y -155.930,Z 1887.279,A 0.000,B 0.000,C 90.000,E1 230.194} C_DIS
LIN {X -0.093,Y -152.182,Z 1887.254,A 0.000,B 0.000,C 90.000,E1 225.729} C_DIS
LIN {X 0.031,Y -150.429,Z 1887.239,A 0.000,B 0.000,C 90.000,E1 222.975} C_DIS
LIN {X -0.044,Y -147.156,Z 1887.214,A 0.000,B 0.000,C 90.000,E1 218.463} C_DIS
LIN {X -0.076,Y -145.171,Z 1887.193,A 0.000,B 0.000,C 90.000,E1 214.818} C_DIS
LIN {X -0.041,Y -142.322,Z 1887.163,A 0.000,B 0.000,C 90.000,E1 209.283} C_DIS
LIN {X 0.080,Y -141.710,Z 1887.152,A 0.000,B 0.000,C 90.000,E1 207.385} C_DIS
LIN {X 0.002,Y -139.471,Z 1887.116,A 0.000,B 0.000,C 90.000,E1 200.918} C_DIS
LIN {X 0.056,Y -139.203,Z 1887.106,A 0.000,B 0.000,C 90.000,E1 199.033} C_DIS
LIN {X -0.017,Y -138.329,Z 1887.054,A 0.000,B 0.000,C 90.000,E1 189.726} C_DIS
LIN {X -0.014,Y -139.440,Z 1887.007,A 0.000,B 0.000,C 90.000,E1 181.318} C_DIS
LIN {X 0.066,Y -140.972,Z 1886.976,A 0.000,B 0.000,C 90.000,E1 175.698} C_DIS
LIN {X 0.016,Y -142.728,Z 1886.956,A 0.000,B 0.000,C 90.000,E1 172.008} C_DIS
LIN {X -0.026,Y -145.114,Z 1886.930,A 0.000,B 0.000,C 90.000,E1 167.409} C_DIS
LIN {X -0.032,Y -147.737,Z 1886.910,A 0.000,B 0.000,C 90.000,E1 163.740} C_DIS
LIN {X 0.049,Y -150.402,Z 1886.889,A 0.000,B 0.000,C 90.000,E1 160.061} C_DIS
LIN {X -0.076,Y -153.838,Z 1886.869,A 0.000,B 0.000,C 90.000,E1 156.485} C_DIS
LIN {X -0.017,Y -157.249,Z 1886.849,A 0.000,B 0.000,C 90.000,E1 152.871} C_DIS
LIN {X -0.077,Y -161.422,Z 1886.829,A 0.000,B 0.000,C 90.000,E1 149.331} C_DIS
LIN {X -0.068,Y -165.622,Z 1886.810,A 0.000,B 0.000,C 90.000,E1 145.801} C_DIS
LIN {X 0.053,Y -170.551,Z 1886.791,A 0.000,B 0.000,C 90.000,E1 142.271} C_DIS
LIN {X -0.040,Y -175.429,Z 1886.771,A 0.000,B 0.000,C 90.000,E1 138.852} C_DIS
LIN {X 0.077,Y -181.053,Z 1886.752,A 0.000,B 0.000,C 90.000,E1 135.405} C_DIS
LIN {X -0.057,Y -186.489,Z 1886.734,A 0.000,B 0.000,C 90.000,E1 132.081} C_DIS
LIN {X 0.011,Y -191.111,Z 1886.720,A 0.000,B 0.000,C 90.000,E1 129.564} C_DIS
LIN {X -0.069,Y -196.905,Z 1886.702,A 0.000,B 0.000,C 90.000,E1 126.297} C_DIS
LIN {X -0.038,Y -200.165,Z 1886.693,A 0.000,B 0.000,C 90.000,E1 124.659} C_DIS
LIN {X 0.124,Y -207.662,Z 1886.670,A 0.000,B 0.000,C 90.000,E1 120.590} C_DIS
LIN {X 0.026,Y -210.853,Z 1886.661,A 0.000,B 0.000,C 90.000,E1 119.027} C_DIS
LIN {X -0.059,Y -216.710,Z 1886.644,A 0.000,B 0.000,C 90.000,E1 115.899} C_DIS
LIN {X -0.045,Y -219.776,Z 1886.635,A 0.000,B 0.000,C 90.000,E1 114.335} C_DIS
LIN {X -0.015,Y -224.118,Z 1886.621,A 0.000,B 0.000,C 90.000,E1 111.844} C_DIS
LIN {X -0.051,Y -283.392,Z 1886.621,A 0.000,B 0.000,C 90.000,E1 111.844} C_DIS
LIN {X 0.102,Y -288.369,Z 1886.620,A 0.000,B 0.000,C 90.000,E1 111.663} C_DIS
LIN {X -0.013,Y -290.578,Z 1886.620,A 0.000,B 0.000,C 90.000,E1 111.535} C_DIS
LIN {X 0.027,Y -293.575,Z 1886.618,A 0.000,B 0.000,C 90.000,E1 111.227} C_DIS
LIN {X -0.014,Y -297.256,Z 1886.615,A 0.000,B 0.000,C 90.000,E1 110.663} C_DIS
LIN {X -0.106,Y -310.592,Z 1886.602,A 0.000,B 0.000,C 90.000,E1 108.362} C_DIS
LIN {X 0.017,Y -325.297,Z 1886.589,A 0.000,B 0.000,C 90.000,E1 106.079} C_DIS
LIN {X 0.010,Y -339.092,Z 1886.579,A 0.000,B 0.000,C 90.000,E1 104.189} C_DIS
LIN {X -0.066,Y -354.080,Z 1886.569,A 0.000,B 0.000,C 90.000,E1 102.355} C_DIS
LIN {X 0.067,Y -372.502,Z 1886.557,A 0.000,B 0.000,C 90.000,E1 100.310} C_DIS
LIN {X 0.161,Y -391.399,Z 1886.547,A 0.000,B 0.000,C 90.000,E1 98.454} C_DIS
LIN {X 0.188,Y -410.635,Z 1886.538,A 0.000,B 0.000,C 90.000,E1 96.777} C_DIS
LIN {X 0.117,Y -433.034,Z 1886.528,A 0.000,B 0.000,C 90.000,E1 95.049} C_DIS
LIN {X 0.093,Y -438.692,Z 1886.526,A 0.000,B 0.000,C 90.000,E1 94.645} C_DIS
LIN {X -0.137,Y -441.105,Z 1886.525,A 0.000,B 0.000,C 90.000,E1 94.473} C_DIS
LIN {X -0.048,Y -444.670,Z 1886.522,A 0.000,B 0.000,C 90.000,E1 94.012} C_DIS
LIN {X 0.124,Y -446.077,Z 1886.521,A 0.000,B 0.000,C 90.000,E1 93.726} C_DIS
LIN {X -0.149,Y -447.131,Z 1886.519,A 0.000,B 0.000,C 90.000,E1 93.498} C_DIS
LIN {X -0.194,Y -448.377,Z 1886.516,A 0.000,B 0.000,C 90.000,E1 92.980} C_DIS
LIN {X 0.194,Y -448.650,Z 1886.514,A 0.000,B 0.000,C 90.000,E1 92.407} C_DIS
LIN {X 0.143,Y -447.995,Z 1886.511,A 0.000,B 0.000,C 90.000,E1 91.892} C_DIS
LIN {X 0.106,Y -446.314,Z 1886.508,A 0.000,B 0.000,C 90.000,E1 91.375} C_DIS
LIN {X -0.143,Y -444.998,Z 1886.506,A 0.000,B 0.000,C 90.000,E1 91.146} C_DIS
LIN {X -0.205,Y -433.495,Z 1886.496,A 0.000,B 0.000,C 90.000,E1 89.312} C_DIS
LIN {X 0.106,Y -425.172,Z 1886.489,A 0.000,B 0.000,C 90.000,E1 87.936} C_DIS
LIN {X 0.182,Y -411.708,Z 1886.477,A 0.000,B 0.000,C 90.000,E1 85.755} C_DIS
LIN {X -0.160,Y -401.539,Z 1886.467,A 0.000,B 0.000,C 90.000,E1 84.147} C_DIS
LIN {X -0.178,Y -389.577,Z 1886.456,A 0.000,B 0.000,C 90.000,E1 82.186} C_DIS
LIN {X 0.040,Y -377.667,Z 1886.445,A 0.000,B 0.000,C 90.000,E1 80.151} C_DIS
LIN {X 0.021,Y -361.029,Z 1886.429,A 0.000,B 0.000,C 90.000,E1 77.229} C_DIS
LIN {X 0.099,Y -345.434,Z 1886.412,A 0.000,B 0.000,C 90.000,E1 74.212} C_DIS
LIN {X 0.032,Y -333.467,Z 1886.399,A 0.000,B 0.000,C 90.000,E1 71.764} C_DIS
LIN {X -0.010,Y -321.770,Z 1886.385,A 0.000,B 0.000,C 90.000,E1 69.263} C_DIS
LIN {X 0.113,Y -309.149,Z 1886.369,A 0.000,B 0.000,C 90.000,E1 66.357} C_DIS
LIN {X 0.081,Y -299.624,Z 1886.356,A 0.000,B 0.000,C 90.000,E1 64.076} C_DIS
LIN {X -0.040,Y -287.565,Z 1886.339,A 0.000,B 0.000,C 90.000,E1 61.101} C_DIS
LIN {X -0.129,Y -278.132,Z 1886.326,A 0.000,B 0.000,C 90.000,E1 58.742} C_DIS
LIN {X 0.003,Y -268.654,Z 1886.313,A 0.000,B 0.000,C 90.000,E1 56.294} C_DIS
LIN {X -0.049,Y -260.444,Z 1886.301,A 0.000,B 0.000,C 90.000,E1 54.196} C_DIS
LIN {X -0.077,Y -250.837,Z 1886.287,A 0.000,B 0.000,C 90.000,E1 51.698} C_DIS
LIN {X -0.038,Y -241.282,Z 1886.273,A 0.000,B 0.000,C 90.000,E1 49.138} C_DIS
LIN {X 0.070,Y -230.634,Z 1886.256,A 0.000,B 0.000,C 90.000,E1 46.134} C_DIS
LIN {X 0.058,Y -220.430,Z 1886.240,A 0.000,B 0.000,C 90.000,E1 43.095} C_DIS
LIN {X -0.029,Y -210.812,Z 1886.222,A 0.000,B 0.000,C 90.000,E1 40.011} C_DIS
LIN {X -0.125,Y -202.038,Z 1886.205,A 0.000,B 0.000,C 90.000,E1 36.870} C_DIS
LIN {X -0.049,Y -194.073,Z 1886.187,A 0.000,B 0.000,C 90.000,E1 33.627} C_DIS
LIN {X -0.008,Y -186.853,Z 1886.168,A 0.000,B 0.000,C 90.000,E1 30.335} C_DIS
LIN {X -0.003,Y -180.335,Z 1886.150,A 0.000,B 0.000,C 90.000,E1 27.001} C_DIS
LIN {X 0.015,Y -175.916,Z 1886.136,A 0.000,B 0.000,C 90.000,E1 24.463} C_DIS
LIN {X 0.018,Y -170.770,Z 1886.117,A 0.000,B 0.000,C 90.000,E1 21.046} C_DIS
LIN {X 0.034,Y -166.397,Z 1886.098,A 0.000,B 0.000,C 90.000,E1 17.583} C_DIS
LIN {X -0.048,Y -162.825,Z 1886.078,A 0.000,B 0.000,C 90.000,E1 14.120} C_DIS
LIN {X 0.076,Y -159.212,Z 1886.054,A 0.000,B 0.000,C 90.000,E1 9.670} C_DIS
LIN {X 0.012,Y -156.385,Z 1886.024,A 0.000,B 0.000,C 90.000,E1 4.359} C_DIS
LIN {X -0.015,Y -154.159,Z 1885.982,A 0.000,B 0.000,C 90.000,E1 356.846} C_DIS
LIN {X -0.001,Y -155.123,Z 1885.923,A 0.000,B 0.000,C 90.000,E1 346.061} C_DIS
LIN {X 0.036,Y -157.420,Z 1885.893,A 0.000,B 0.000,C 90.000,E1 340.678} C_DIS
LIN {X 0.033,Y -160.562,Z 1885.868,A 0.000,B 0.000,C 90.000,E1 336.230} C_DIS
LIN {X 0.044,Y -164.002,Z 1885.848,A 0.000,B 0.000,C 90.000,E1 332.692} C_DIS
LIN {X 0.002,Y -168.445,Z 1885.829,A 0.000,B 0.000,C 90.000,E1 329.203} C_DIS
LIN {X -0.081,Y -172.409,Z 1885.814,A 0.000,B 0.000,C 90.000,E1 326.628} C_DIS
LIN {X -0.044,Y -176.953,Z 1885.800,A 0.000,B 0.000,C 90.000,E1 324.036} C_DIS
LIN {X -0.006,Y -179.542,Z 1885.793,A 0.000,B 0.000,C 90.000,E1 322.718} C_DIS
LIN {X -0.027,Y -185.395,Z 1885.793,A 0.000,B 0.000,C 90.000,E1 322.718} C_DIS
LIN {X -0.005,Y -186.679,Z 1885.792,A 0.000,B 0.000,C 90.000,E1 322.637} C_DIS
LIN {X 0.003,Y -188.669,Z 1885.791,A 0.000,B 0.000,C 90.000,E1 322.316} C_DIS
LIN {X -0.006,Y -190.335,Z 1885.788,A 0.000,B 0.000,C 90.000,E1 321.904} C_DIS
LIN {X -0.052,Y -192.920,Z 1885.784,A 0.000,B 0.000,C 90.000,E1 321.090} C_DIS
LIN {X 0.048,Y -196.079,Z 1885.777,A 0.000,B 0.000,C 90.000,E1 319.828} C_DIS
LIN {X -0.112,Y -199.766,Z 1885.768,A 0.000,B 0.000,C 90.000,E1 318.243} C_DIS
LIN {X -0.054,Y -206.935,Z 1885.750,A 0.000,B 0.000,C 90.000,E1 315.000} C_DIS
LIN {X -0.030,Y -212.983,Z 1885.737,A 0.000,B 0.000,C 90.000,E1 312.609} C_DIS
LIN {X 0.026,Y -217.680,Z 1885.728,A 0.000,B 0.000,C 90.000,E1 311.024} C_DIS
LIN {X 0.056,Y -221.813,Z 1885.721,A 0.000,B 0.000,C 90.000,E1 309.850} C_DIS
LIN {X 0.021,Y -229.632,Z 1885.711,A 0.000,B 0.000,C 90.000,E1 307.935} C_DIS
LIN {X -0.038,Y -241.882,Z 1885.696,A 0.000,B 0.000,C 90.000,E1 305.311} C_DIS
LIN {X -0.108,Y -255.065,Z 1885.682,A 0.000,B 0.000,C 90.000,E1 302.752} C_DIS
LIN {X 0.035,Y -265.131,Z 1885.672,A 0.000,B 0.000,C 90.000,E1 300.924} C_DIS
LIN {X 0.135,Y -282.471,Z 1885.656,A 0.000,B 0.000,C 90.000,E1 298.103} C_DIS
LIN {X 0.069,Y -293.728,Z 1885.647,A 0.000,B 0.000,C 90.000,E1 296.411} C_DIS
LIN {X -0.077,Y -307.062,Z 1885.636,A 0.000,B 0.000,C 90.000,E1 294.439} C_DIS
LIN {X 0.142,Y -318.051,Z 1885.627,A 0.000,B 0.000,C 90.000,E1 292.770} C_DIS
LIN {X -0.180,Y -328.615,Z 1885.618,A 0.000,B 0.000,C 90.000,E1 291.227} C_DIS
LIN {X -0.012,Y -336.673,Z 1885.611,A 0.000,B 0.000,C 90.000,E1 289.939} C_DIS
LIN {X -0.168,Y -342.351,Z 1885.606,A 0.000,B 0.000,C 90.000,E1 289.033} C_DIS
LIN {X 0.161,Y -347.614,Z 1885.600,A 0.000,B 0.000,C 90.000,E1 288.055} C_DIS
